LIN {X 0,Y 300.031,Z 474.405,A -85,B 0,C 180,E1 -16672.737,E2 -16672.737} C_VEL
LIN {X 0,Y 302.31,Z 463.313,A -85,B 0,C 180,E1 -16674.577,E2 -16674.577} C_VEL
LIN {X 0,Y 303.513,Z 452.468,A -85,B 0,C 180,E1 -16676.262,E2 -16676.262} C_VEL
LIN {X 0,Y 303.68,Z 440.033,A -85,B 0,C 180,E1 -16678.173,E2 -16678.173} C_VEL
LIN {X 0,Y 303.07,Z 428.896,A -85,B 0,C 180,E1 -16679.914,E2 -16679.914} C_VEL
LIN {X 0,Y 301.506,Z 416.977,A -85,B 0,C 180,E1 -16681.946,E2 -16681.946} C_VEL
LIN {X 0,Y 300.427,Z 410.712,A -85,B 0,C 180,E1 -16683.112,E2 -16683.112} C_VEL
LIN {X 0,Y 299.765,Z 406.041,A -85,B 0,C 180,E1 -16683.974,E2 -16683.974} C_VEL
LIN {X 0,Y 298.458,Z 400.385,A -85,B 0,C 180,E1 -16685.221,E2 -16685.221} C_VEL
LIN {X 0,Y 298.188,Z 398.22,A -85,B 0,C 180,E1 -16685.654,E2 -16685.654} C_VEL
LIN {X 0,Y 296.755,Z 392.365,A -85,B 0,C 180,E1 -16687.15,E2 -16687.15} C_VEL
LIN {X 0,Y 296.569,Z 389.678,A -85,B 0,C 180,E1 -16687.712,E2 -16687.712} C_VEL
LIN {X 0,Y 297.108,Z 387.807,A -85,B 0,C 180,E1 -16688.684,E2 -16688.684} C_VEL
LIN {X 0,Y 296.56,Z 383.262,A -85,B 0,C 180,E1 -16691.572,E2 -16691.572} C_VEL
LIN {X 0,Y 295.752,Z 379.256,A -85,B 0,C 180,E1 -16694.529,E2 -16694.529} C_VEL
LIN {X 0,Y 294.903,Z 375.161,A -85,B 0,C 180,E1 -16698.142,E2 -16698.142} C_VEL
LIN {X 0,Y 294.504,Z 373.34,A -85,B 0,C 180,E1 -16700.14,E2 -16700.14} C_VEL
LIN {X 0,Y 295.68,Z 374.442,A -85,B 0,C 180,E1 -16701.83,E2 -16701.83} C_VEL
LIN {X 0,Y 298.13,Z 375.151,A -85,B 0,C 180,E1 -16703.889,E2 -16703.889} C_VEL
LIN {X 0,Y 300.781,Z 377.325,A -85,B 0,C 180,E1 -16705.89,E2 -16705.89} C_VEL
LIN {X 0,Y 303.781,Z 380.298,A -85,B 0,C 180,E1 -16707.852,E2 -16707.852} C_VEL
LIN {X 0,Y 306.859,Z 384.143,A -85,B 0,C 180,E1 -16709.744,E2 -16709.744} C_VEL
LIN {X 0,Y 308.626,Z 387.569,A -85,B 0,C 180,E1 -16710.989,E2 -16710.989} C_VEL
LIN {X 0,Y 311.017,Z 394.757,A -85,B 0,C 180,E1 -16713.132,E2 -16713.132} C_VEL
LIN {X 0,Y 312.633,Z 402.039,A -85,B 0,C 180,E1 -16715.127,E2 -16715.127} C_VEL
LIN {X 0,Y 312.849,Z 403.656,A -85,B 0,C 180,E1 -16715.556,E2 -16715.556} C_VEL
LIN {X 0,Y 312.16,Z 406.591,A -85,B 0,C 180,E1 -16716.093,E2 -16716.093} C_VEL
LIN {X 0,Y 308.955,Z 416.302,A -85,B 0,C 180,E1 -16717.955,E2 -16717.955} C_VEL
LIN {X 0,Y 305.609,Z 425.337,A -85,B 0,C 180,E1 -16720.172,E2 -16720.172} C_VEL
LIN {X 0,Y 303.022,Z 431.501,A -85,B 0,C 180,E1 -16722.067,E2 -16722.067} C_VEL
LIN {X 0,Y 300.27,Z 437.333,A -85,B 0,C 180,E1 -16724.385,E2 -16724.385} C_VEL
LIN {X 0,Y 298.323,Z 441.092,A -85,B 0,C 180,E1 -16726.374,E2 -16726.374} C_VEL
LIN {X 0,Y 297.094,Z 443.088,A -85,B 0,C 180,E1 -16727.707,E2 -16727.707} C_VEL
LIN {X 0,Y 296.038,Z 444.641,A -85,B 0,C 180,E1 -16729.052,E2 -16729.052} C_VEL
LIN {X 0,Y 294.259,Z 446.525,A -85,B 0,C 180,E1 -16731.761,E2 -16731.761} C_VEL
LIN {X 0,Y 293.551,Z 446.906,A -85,B 0,C 180,E1 -16733.125,E2 -16733.125} C_VEL
LIN {X 0,Y 292.972,Z 446.863,A -85,B 0,C 180,E1 -16734.494,E2 -16734.494} C_VEL
LIN {X 0,Y 292.076,Z 445.605,A -85,B 0,C 180,E1 -16737.241,E2 -16737.241} C_VEL
LIN {X 0,Y 291.848,Z 444.386,A -85,B 0,C 180,E1 -16738.62,E2 -16738.62} C_VEL
LIN {X 0,Y 291.592,Z 441.785,A -85,B 0,C 180,E1 -16740.69,E2 -16740.69} C_VEL
LIN {X 0,Y 291.444,Z 438.224,A -85,B 0,C 180,E1 -16742.764,E2 -16742.764} C_VEL
LIN {X 0,Y 291.319,Z 435.273,A -85,B 0,C 180,E1 -16744.15,E2 -16744.15} C_VEL
LIN {X 0,Y 291.852,Z 429.89,A -85,B 0,C 180,E1 -16746.221,E2 -16746.221} C_VEL
LIN {X 0,Y 292.35,Z 422.074,A -85,B 0,C 180,E1 -16748.641,E2 -16748.641} C_VEL
LIN {X 0,Y 293.021,Z 413.88,A -85,B 0,C 180,E1 -16750.677,E2 -16750.677} C_VEL
LIN {X 0,Y 293.763,Z 403.548,A -85,B 0,C 180,E1 -16752.785,E2 -16752.785} C_VEL
LIN {X 0,Y 294.713,Z 393.16,A -85,B 0,C 180,E1 -16754.501,E2 -16754.501} C_VEL
LIN {X 0,Y 295.536,Z 381.754,A -85,B 0,C 180,E1 -16756.048,E2 -16756.048} C_VEL
LIN {X 0,Y 295.769,Z 377.353,A -85,B 0,C 180,E1 -16756.567,E2 -16756.567} C_VEL
LIN {X 0,Y 293.177,Z 366.301,A -85,B 0,C 180,E1 -16757.828,E2 -16757.828} C_VEL
LIN {X 0,Y 291.511,Z 359.165,A -85,B 0,C 180,E1 -16758.538,E2 -16758.538} C_VEL
LIN {X 0,Y 291.436,Z 359.181,A -85,B 0,C 180,E1 -16763.598,E2 -16763.598} C_VEL
LIN {X 0,Y 291.425,Z 359.184,A -85,B 0,C 180,E1 -16767.271,E2 -16767.271} C_VEL
LIN {X 0,Y 291.339,Z 359.193,A -85,B 0,C 180,E1 -16770.436,E2 -16770.436} C_VEL
LIN {X 0,Y 291.347,Z 359.19,A -85,B 0,C 180,E1 -16773.698,E2 -16773.698} C_VEL
LIN {X 0,Y 291.4,Z 359.186,A -85,B 0,C 180,E1 -16777.26,E2 -16777.26} C_VEL
LIN {X 0,Y 291.378,Z 359.19,A -85,B 0,C 180,E1 -16780.635,E2 -16780.635} C_VEL
LIN {X 0,Y 291.325,Z 359.195,A -85,B 0,C 180,E1 -16784.395,E2 -16784.395} C_VEL
LIN {X 0,Y 291.328,Z 359.196,A -85,B 0,C 180,E1 -16788.404,E2 -16788.404} C_VEL
LIN {X 0,Y 291.365,Z 359.189,A -85,B 0,C 180,E1 -16791.16,E2 -16791.16} C_VEL
LIN {X 0,Y 291.386,Z 359.191,A -85,B 0,C 180,E1 -16794.629,E2 -16794.629} C_VEL
LIN {X 0,Y 291.371,Z 359.189,A -85,B 0,C 180,E1 -16797.95,E2 -16797.95} C_VEL
LIN {X 0,Y 291.378,Z 359.187,A -85,B 0,C 180,E1 -16801.158,E2 -16801.158} C_VEL
LIN {X 0,Y 291.415,Z 359.186,A -85,B 0,C 180,E1 -16804.272,E2 -16804.272} C_VEL
LIN {X 0,Y 291.391,Z 359.185,A -85,B 0,C 180,E1 -16807.3,E2 -16807.3} C_VEL
LIN {X 0,Y 291.464,Z 359.18,A -85,B 0,C 180,E1 -16810.271,E2 -16810.271} C_VEL
LIN {X 0,Y 291.556,Z 359.167,A -85,B 0,C 180,E1 -16814.624,E2 -16814.624} C_VEL
LIN {X 0,Y 291.536,Z 359.167,A -85,B 0,C 180,E1 -16818.881,E2 -16818.881} C_VEL
LIN {X 0,Y 291.688,Z 359.15,A -85,B 0,C 180,E1 -16821.688,E2 -16821.688} C_VEL
LIN {X 0,Y 291.628,Z 359.157,A -85,B 0,C 180,E1 -16824.468,E2 -16824.468} C_VEL
LIN {X 0,Y 291.889,Z 359.124,A -85,B 0,C 180,E1 -16828.62,E2 -16828.62} C_VEL
LIN {X 0,Y 291.891,Z 359.124,A -85,B 0,C 180,E1 -16831.38,E2 -16831.38} C_VEL
LIN {X 0,Y 291.736,Z 359.142,A -85,B 0,C 180,E1 -16836.918,E2 -16836.918} C_VEL
LIN {X 0,Y 291.576,Z 359.166,A -85,B 0,C 180,E1 -16839.714,E2 -16839.714} C_VEL
LIN {X 0,Y 291.523,Z 359.172,A -85,B 0,C 180,E1 -16843.95,E2 -16843.95} C_VEL
LIN {X 0,Y 291.488,Z 359.173,A -85,B 0,C 180,E1 -16846.818,E2 -16846.818} C_VEL
LIN {X 0,Y 291.451,Z 359.18,A -85,B 0,C 180,E1 -16849.875,E2 -16849.875} C_VEL
LIN {X 0,Y 291.401,Z 359.185,A -85,B 0,C 180,E1 -16854.205,E2 -16854.205} C_VEL
LIN {X 0,Y 291.421,Z 359.184,A -85,B 0,C 180,E1 -16857.272,E2 -16857.272} C_VEL
LIN {X 0,Y 291.335,Z 359.191,A -85,B 0,C 180,E1 -16860.437,E2 -16860.437} C_VEL
LIN {X 0,Y 291.346,Z 359.194,A -85,B 0,C 180,E1 -16863.699,E2 -16863.699} C_VEL
LIN {X 0,Y 291.4,Z 359.188,A -85,B 0,C 180,E1 -16867.26,E2 -16867.26} C_VEL
LIN {X 0,Y 291.402,Z 359.184,A -85,B 0,C 180,E1 -16870.631,E2 -16870.631} C_VEL
LIN {X 0,Y 291.354,Z 359.19,A -85,B 0,C 180,E1 -16874.39,E2 -16874.39} C_VEL
LIN {X 0,Y 291.333,Z 359.192,A -85,B 0,C 180,E1 -16878.404,E2 -16878.404} C_VEL
LIN {X 0,Y 291.35,Z 359.196,A -85,B 0,C 180,E1 -16881.158,E2 -16881.158} C_VEL
LIN {X 0,Y 291.363,Z 359.19,A -85,B 0,C 180,E1 -16884.627,E2 -16884.627} C_VEL
LIN {X 0,Y 291.374,Z 359.187,A -85,B 0,C 180,E1 -16887.951,E2 -16887.951} C_VEL
LIN {X 0,Y 291.386,Z 359.189,A -85,B 0,C 180,E1 -16891.159,E2 -16891.159} C_VEL
LIN {X 0,Y 291.42,Z 359.181,A -85,B 0,C 180,E1 -16894.272,E2 -16894.272} C_VEL
LIN {X 0,Y 291.385,Z 359.188,A -85,B 0,C 180,E1 -16897.3,E2 -16897.3} C_VEL
LIN {X 0,Y 291.461,Z 359.177,A -85,B 0,C 180,E1 -16900.271,E2 -16900.271} C_VEL
LIN {X 0,Y 291.559,Z 359.168,A -85,B 0,C 180,E1 -16904.624,E2 -16904.624} C_VEL
LIN {X 0,Y 291.541,Z 359.17,A -85,B 0,C 180,E1 -16908.881,E2 -16908.881} C_VEL
LIN {X 0,Y 291.713,Z 359.144,A -85,B 0,C 180,E1 -16911.689,E2 -16911.689} C_VEL
LIN {X 0,Y 291.634,Z 359.159,A -85,B 0,C 180,E1 -16914.469,E2 -16914.469} C_VEL
LIN {X 0,Y 291.893,Z 359.126,A -85,B 0,C 180,E1 -16918.621,E2 -16918.621} C_VEL
LIN {X 0,Y 291.895,Z 359.122,A -85,B 0,C 180,E1 -16921.38,E2 -16921.38} C_VEL
LIN {X 0,Y 291.727,Z 359.144,A -85,B 0,C 180,E1 -16926.919,E2 -16926.919} C_VEL
LIN {X 0,Y 291.576,Z 359.162,A -85,B 0,C 180,E1 -16929.714,E2 -16929.714} C_VEL
LIN {X 0,Y 291.526,Z 359.168,A -85,B 0,C 180,E1 -16931.342,E2 -16931.342} C_VEL
LIN {X 0,Y 290.829,Z 359.259,A -85,B 0,C 180,E1 -16932.496,E2 -16932.496} C_VEL
LIN {X 0,Y 287.986,Z 359.613,A -85,B 0,C 180,E1 -16934.375,E2 -16934.375} C_VEL
LIN {X 0,Y 285.575,Z 359.913,A -85,B 0,C 180,E1 -16935.9,E2 -16935.9} C_VEL
LIN {X 0,Y 284.515,Z 360.041,A -85,B 0,C 180,E1 -16937.081,E2 -16937.081} C_VEL
LIN {X 0,Y 284.414,Z 360.052,A -85,B 0,C 180,E1 -16937.481,E2 -16937.481} C_VEL
LIN {X 0,Y 284.383,Z 360.063,A -85,B 0,C 180,E1 -16940.242,E2 -16940.242} C_VEL
LIN {X 0,Y 284.373,Z 360.062,A -85,B 0,C 180,E1 -16943.876,E2 -16943.876} C_VEL
LIN {X 0,Y 284.401,Z 360.055,A -85,B 0,C 180,E1 -16947.174,E2 -16947.174} C_VEL
LIN {X 0,Y 284.3,Z 360.069,A -85,B 0,C 180,E1 -16951.274,E2 -16951.274} C_VEL
LIN {X 0,Y 284.365,Z 360.061,A -85,B 0,C 180,E1 -16955.354,E2 -16955.354} C_VEL
LIN {X 0,Y 284.327,Z 360.068,A -85,B 0,C 180,E1 -16958.167,E2 -16958.167} C_VEL
LIN {X 0,Y 284.35,Z 360.119,A -85,B 0,C 180,E1 -16961.862,E2 -16961.862} C_VEL
LIN {X 0,Y 285.952,Z 368.508,A -85,B 0,C 180,E1 -16966.021,E2 -16966.021} C_VEL
LIN {X 0,Y 287.637,Z 376.818,A -85,B 0,C 180,E1 -16969.956,E2 -16969.956} C_VEL
LIN {X 0,Y 288.32,Z 381.031,A -85,B 0,C 180,E1 -16971.889,E2 -16971.889} C_VEL
LIN {X 0,Y 287.289,Z 387.971,A -85,B 0,C 180,E1 -16974.908,E2 -16974.908} C_VEL
LIN {X 0,Y 285.874,Z 397.284,A -85,B 0,C 180,E1 -16978.917,E2 -16978.917} C_VEL
LIN {X 0,Y 284.593,Z 408.243,A -85,B 0,C 180,E1 -16983.608,E2 -16983.608} C_VEL
LIN {X 0,Y 283.665,Z 419.379,A -85,B 0,C 180,E1 -16988.374,E2 -16988.374} C_VEL
LIN {X 0,Y 284.085,Z 432.923,A -85,B 0,C 180,E1 -16989.168,E2 -16989.168} C_VEL
LIN {X 0,Y 284.692,Z 446.489,A -85,B 0,C 180,E1 -16990.251,E2 -16990.251} C_VEL
LIN {X 0,Y 285.479,Z 460.384,A -85,B 0,C 180,E1 -16991.706,E2 -16991.706} C_VEL
LIN {X 0,Y 286.008,Z 471.143,A -85,B 0,C 180,E1 -16993.105,E2 -16993.105} C_VEL
LIN {X 0,Y 285.619,Z 477.09,A -85,B 0,C 180,E1 -16994.016,E2 -16994.016} C_VEL
LIN {X 0,Y 284.793,Z 486.616,A -85,B 0,C 180,E1 -16995.713,E2 -16995.713} C_VEL
LIN {X 0,Y 284.282,Z 494.949,A -85,B 0,C 180,E1 -16997.507,E2 -16997.507} C_VEL
LIN {X 0,Y 283.889,Z 503.067,A -85,B 0,C 180,E1 -16999.66,E2 -16999.66} C_VEL
LIN {X 0,Y 283.879,Z 510.11,A -85,B 0,C 180,E1 -17002.007,E2 -17002.007} C_VEL
LIN {X 0,Y 284.172,Z 515.473,A -85,B 0,C 180,E1 -17004.323,E2 -17004.323} C_VEL
LIN {X 0,Y 284.473,Z 519.112,A -85,B 0,C 180,E1 -17006.459,E2 -17006.459} C_VEL
LIN {X 0,Y 284.734,Z 521.591,A -85,B 0,C 180,E1 -17008.586,E2 -17008.586} C_VEL
LIN {X 0,Y 284.939,Z 522.63,A -85,B 0,C 180,E1 -17010,E2 -17010} C_VEL
LIN {X 0,Y 284.508,Z 523.101,A -85,B 0,C 180,E1 -17011.415,E2 -17011.415} C_VEL
LIN {X 0,Y 283.776,Z 522.795,A -85,B 0,C 180,E1 -17014.261,E2 -17014.261} C_VEL
LIN {X 0,Y 283.234,Z 520.886,A -85,B 0,C 180,E1 -17017.002,E2 -17017.002} C_VEL
LIN {X 0,Y 283.044,Z 518.199,A -85,B 0,C 180,E1 -17019.288,E2 -17019.288} C_VEL
LIN {X 0,Y 283.523,Z 513.371,A -85,B 0,C 180,E1 -17022.163,E2 -17022.163} C_VEL
LIN {X 0,Y 284.82,Z 506.896,A -85,B 0,C 180,E1 -17025.016,E2 -17025.016} C_VEL
LIN {X 0,Y 286.666,Z 499.719,A -85,B 0,C 180,E1 -17027.477,E2 -17027.477} C_VEL
LIN {X 0,Y 289.388,Z 491.01,A -85,B 0,C 180,E1 -17029.877,E2 -17029.877} C_VEL
LIN {X 0,Y 291.945,Z 482.139,A -85,B 0,C 180,E1 -17031.909,E2 -17031.909} C_VEL
LIN {X 0,Y 294.468,Z 471.795,A -85,B 0,C 180,E1 -17033.937,E2 -17033.937} C_VEL
LIN {X 0,Y 296.624,Z 461.632,A -85,B 0,C 180,E1 -17035.679,E2 -17035.679} C_VEL
LIN {X 0,Y 297.814,Z 450.071,A -85,B 0,C 180,E1 -17037.589,E2 -17037.589} C_VEL
LIN {X 0,Y 298.028,Z 437.389,A -85,B 0,C 180,E1 -17039.684,E2 -17039.684} C_VEL
LIN {X 0,Y 297.318,Z 425.925,A -85,B 0,C 180,E1 -17041.682,E2 -17041.682} C_VEL
LIN {X 0,Y 296.145,Z 415.72,A -85,B 0,C 180,E1 -17043.636,E2 -17043.636} C_VEL
LIN {X 0,Y 295.085,Z 408.633,A -85,B 0,C 180,E1 -17045.142,E2 -17045.142} C_VEL
LIN {X 0,Y 294.416,Z 403.054,A -85,B 0,C 180,E1 -17046.359,E2 -17046.359} C_VEL
LIN {X 0,Y 293.422,Z 397.739,A -85,B 0,C 180,E1 -17047.776,E2 -17047.776} C_VEL
LIN {X 0,Y 293.175,Z 394.527,A -85,B 0,C 180,E1 -17048.556,E2 -17048.556} C_VEL
LIN {X 0,Y 292.293,Z 391.653,A -85,B 0,C 180,E1 -17049.698,E2 -17049.698} C_VEL
LIN {X 0,Y 290.67,Z 386.21,A -85,B 0,C 180,E1 -17052.61,E2 -17052.61} C_VEL
LIN {X 0,Y 290.204,Z 383.651,A -85,B 0,C 180,E1 -17054.613,E2 -17054.613} C_VEL
LIN {X 0,Y 290.482,Z 381.502,A -85,B 0,C 180,E1 -17057.356,E2 -17057.356} C_VEL
LIN {X 0,Y 292.166,Z 380.152,A -85,B 0,C 180,E1 -17060.332,E2 -17060.332} C_VEL
LIN {X 0,Y 293.486,Z 381.114,A -85,B 0,C 180,E1 -17062.208,E2 -17062.208} C_VEL
LIN {X 0,Y 294.854,Z 381.369,A -85,B 0,C 180,E1 -17063.424,E2 -17063.424} C_VEL
LIN {X 0,Y 297.578,Z 383.63,A -85,B 0,C 180,E1 -17065.752,E2 -17065.752} C_VEL
LIN {X 0,Y 299.931,Z 386.143,A -85,B 0,C 180,E1 -17067.518,E2 -17067.518} C_VEL
LIN {X 0,Y 302.454,Z 389.396,A -85,B 0,C 180,E1 -17069.29,E2 -17069.29} C_VEL
LIN {X 0,Y 304.006,Z 392.328,A -85,B 0,C 180,E1 -17070.505,E2 -17070.505} C_VEL
LIN {X 0,Y 305.923,Z 399.005,A -85,B 0,C 180,E1 -17072.647,E2 -17072.647} C_VEL
LIN {X 0,Y 307.232,Z 406.151,A -85,B 0,C 180,E1 -17074.753,E2 -17074.753} C_VEL
LIN {X 0,Y 307.06,Z 408.046,A -85,B 0,C 180,E1 -17075.205,E2 -17075.205} C_VEL
LIN {X 0,Y 304.021,Z 416.608,A -85,B 0,C 180,E1 -17076.859,E2 -17076.859} C_VEL
LIN {X 0,Y 300.855,Z 424.65,A -85,B 0,C 180,E1 -17078.772,E2 -17078.772} C_VEL
LIN {X 0,Y 297.983,Z 431.197,A -85,B 0,C 180,E1 -17080.719,E2 -17080.719} C_VEL
LIN {X 0,Y 295.341,Z 436.536,A -85,B 0,C 180,E1 -17082.695,E2 -17082.695} C_VEL
LIN {X 0,Y 293.066,Z 440.748,A -85,B 0,C 180,E1 -17084.705,E2 -17084.705} C_VEL
LIN {X 0,Y 291.701,Z 443.029,A -85,B 0,C 180,E1 -17086.058,E2 -17086.058} C_VEL
LIN {X 0,Y 290.39,Z 444.878,A -85,B 0,C 180,E1 -17087.419,E2 -17087.419} C_VEL
LIN {X 0,Y 288.333,Z 447.305,A -85,B 0,C 180,E1 -17090.176,E2 -17090.176} C_VEL
LIN {X 0,Y 287.388,Z 447.971,A -85,B 0,C 180,E1 -17091.562,E2 -17091.562} C_VEL
LIN {X 0,Y 286.026,Z 448.048,A -85,B 0,C 180,E1 -17094.359,E2 -17094.359} C_VEL
LIN {X 0,Y 285.062,Z 446.608,A -85,B 0,C 180,E1 -17097.173,E2 -17097.173} C_VEL
LIN {X 0,Y 284.681,Z 443.497,A -85,B 0,C 180,E1 -17100,E2 -17100} C_VEL
LIN {X 0,Y 284.458,Z 440.106,A -85,B 0,C 180,E1 -17102.124,E2 -17102.124} C_VEL
LIN {X 0,Y 284.257,Z 435.712,A -85,B 0,C 180,E1 -17104.253,E2 -17104.253} C_VEL
LIN {X 0,Y 284.802,Z 430.166,A -85,B 0,C 180,E1 -17106.375,E2 -17106.375} C_VEL
LIN {X 0,Y 285.217,Z 423.367,A -85,B 0,C 180,E1 -17108.502,E2 -17108.502} C_VEL
LIN {X 0,Y 285.882,Z 415.183,A -85,B 0,C 180,E1 -17110.593,E2 -17110.593} C_VEL
LIN {X 0,Y 286.644,Z 404.889,A -85,B 0,C 180,E1 -17112.748,E2 -17112.748} C_VEL
LIN {X 0,Y 287.628,Z 394.593,A -85,B 0,C 180,E1 -17114.504,E2 -17114.504} C_VEL
LIN {X 0,Y 288.535,Z 381.958,A -85,B 0,C 180,E1 -17116.267,E2 -17116.267} C_VEL
LIN {X 0,Y 288.781,Z 379.024,A -85,B 0,C 180,E1 -17116.616,E2 -17116.616} C_VEL
LIN {X 0,Y 286.137,Z 367.424,A -85,B 0,C 180,E1 -17117.971,E2 -17117.971} C_VEL
LIN {X 0,Y 284.465,Z 360.045,A -85,B 0,C 180,E1 -17118.734,E2 -17118.734} C_VEL
LIN {X 0,Y 284.372,Z 360.059,A -85,B 0,C 180,E1 -17123.875,E2 -17123.875} C_VEL
LIN {X 0,Y 284.399,Z 360.06,A -85,B 0,C 180,E1 -17127.173,E2 -17127.173} C_VEL
LIN {X 0,Y 284.298,Z 360.071,A -85,B 0,C 180,E1 -17131.274,E2 -17131.274} C_VEL
LIN {X 0,Y 284.363,Z 360.062,A -85,B 0,C 180,E1 -17135.354,E2 -17135.354} C_VEL
LIN {X 0,Y 284.331,Z 360.065,A -85,B 0,C 180,E1 -17138.166,E2 -17138.166} C_VEL
LIN {X 0,Y 284.304,Z 360.067,A -85,B 0,C 180,E1 -17141.87,E2 -17141.87} C_VEL
LIN {X 0,Y 284.266,Z 360.073,A -85,B 0,C 180,E1 -17145.805,E2 -17145.805} C_VEL
LIN {X 0,Y 284.308,Z 360.068,A -85,B 0,C 180,E1 -17150.024,E2 -17150.024} C_VEL
LIN {X 0,Y 284.351,Z 360.062,A -85,B 0,C 180,E1 -17153.617,E2 -17153.617} C_VEL
LIN {X 0,Y 284.308,Z 360.068,A -85,B 0,C 180,E1 -17157.189,E2 -17157.189} C_VEL
LIN {X 0,Y 284.356,Z 360.065,A -85,B 0,C 180,E1 -17160.376,E2 -17160.376} C_VEL
LIN {X 0,Y 284.377,Z 360.059,A -85,B 0,C 180,E1 -17163.586,E2 -17163.586} C_VEL
LIN {X 0,Y 284.37,Z 360.062,A -85,B 0,C 180,E1 -17166.707,E2 -17166.707} C_VEL
LIN {X 0,Y 284.407,Z 360.055,A -85,B 0,C 180,E1 -17171.262,E2 -17171.262} C_VEL
LIN {X 0,Y 284.493,Z 360.048,A -85,B 0,C 180,E1 -17174.459,E2 -17174.459} C_VEL
LIN {X 0,Y 284.488,Z 360.047,A -85,B 0,C 180,E1 -17178.601,E2 -17178.601} C_VEL
LIN {X 0,Y 284.64,Z 360.027,A -85,B 0,C 180,E1 -17181.481,E2 -17181.481} C_VEL
LIN {X 0,Y 284.598,Z 360.034,A -85,B 0,C 180,E1 -17184.331,E2 -17184.331} C_VEL
LIN {X 0,Y 284.856,Z 360,A -85,B 0,C 180,E1 -17188.586,E2 -17188.586} C_VEL
LIN {X 0,Y 284.857,Z 360,A -85,B 0,C 180,E1 -17191.414,E2 -17191.414} C_VEL
LIN {X 0,Y 284.687,Z 360.02,A -85,B 0,C 180,E1 -17197.09,E2 -17197.09} C_VEL
LIN {X 0,Y 284.52,Z 360.045,A -85,B 0,C 180,E1 -17199.957,E2 -17199.957} C_VEL
LIN {X 0,Y 284.482,Z 360.047,A -85,B 0,C 180,E1 -17204.303,E2 -17204.303} C_VEL
LIN {X 0,Y 284.426,Z 360.054,A -85,B 0,C 180,E1 -17207.249,E2 -17207.249} C_VEL
LIN {X 0,Y 284.381,Z 360.059,A -85,B 0,C 180,E1 -17210.242,E2 -17210.242} C_VEL
LIN {X 0,Y 284.37,Z 360.063,A -85,B 0,C 180,E1 -17213.876,E2 -17213.876} C_VEL
LIN {X 0,Y 284.396,Z 360.059,A -85,B 0,C 180,E1 -17217.173,E2 -17217.173} C_VEL
LIN {X 0,Y 284.295,Z 360.072,A -85,B 0,C 180,E1 -17221.275,E2 -17221.275} C_VEL
LIN {X 0,Y 284.363,Z 360.066,A -85,B 0,C 180,E1 -17225.354,E2 -17225.354} C_VEL
LIN {X 0,Y 284.333,Z 360.064,A -85,B 0,C 180,E1 -17228.166,E2 -17228.166} C_VEL
LIN {X 0,Y 284.342,Z 360.064,A -85,B 0,C 180,E1 -17232.141,E2 -17232.141} C_VEL
LIN {X 0,Y 284.298,Z 360.068,A -85,B 0,C 180,E1 -17236.198,E2 -17236.198} C_VEL
LIN {X 0,Y 284.308,Z 360.068,A -85,B 0,C 180,E1 -17240.024,E2 -17240.024} C_VEL
LIN {X 0,Y 284.333,Z 360.065,A -85,B 0,C 180,E1 -17243.614,E2 -17243.614} C_VEL
LIN {X 0,Y 284.31,Z 360.071,A -85,B 0,C 180,E1 -17247.19,E2 -17247.19} C_VEL
LIN {X 0,Y 284.362,Z 360.062,A -85,B 0,C 180,E1 -17250.377,E2 -17250.377} C_VEL
LIN {X 0,Y 284.381,Z 360.058,A -85,B 0,C 180,E1 -17253.587,E2 -17253.587} C_VEL
LIN {X 0,Y 284.37,Z 360.063,A -85,B 0,C 180,E1 -17256.707,E2 -17256.707} C_VEL
LIN {X 0,Y 284.407,Z 360.056,A -85,B 0,C 180,E1 -17261.262,E2 -17261.262} C_VEL
LIN {X 0,Y 284.496,Z 360.046,A -85,B 0,C 180,E1 -17264.459,E2 -17264.459} C_VEL
LIN {X 0,Y 284.493,Z 360.049,A -85,B 0,C 180,E1 -17268.602,E2 -17268.602} C_VEL
LIN {X 0,Y 284.663,Z 360.022,A -85,B 0,C 180,E1 -17271.481,E2 -17271.481} C_VEL
LIN {X 0,Y 284.605,Z 360.033,A -85,B 0,C 180,E1 -17274.332,E2 -17274.332} C_VEL
LIN {X 0,Y 284.859,Z 360.003,A -85,B 0,C 180,E1 -17278.586,E2 -17278.586} C_VEL
LIN {X 0,Y 284.861,Z 359.998,A -85,B 0,C 180,E1 -17281.414,E2 -17281.414} C_VEL
LIN {X 0,Y 284.678,Z 360.021,A -85,B 0,C 180,E1 -17287.091,E2 -17287.091} C_VEL
LIN {X 0,Y 284.521,Z 360.042,A -85,B 0,C 180,E1 -17289.957,E2 -17289.957} C_VEL
LIN {X 0,Y 284.486,Z 360.05,A -85,B 0,C 180,E1 -17294.303,E2 -17294.303} C_VEL
LIN {X 0,Y 284.414,Z 360.052,A -85,B 0,C 180,E1 -17297.481,E2 -17297.481} C_VEL
LIN {X 0,Y 283.687,Z 360.147,A -85,B 0,C 180,E1 -17298.662,E2 -17298.662} C_VEL
LIN {X 0,Y 280.765,Z 360.511,A -85,B 0,C 180,E1 -17300.583,E2 -17300.583} C_VEL
LIN {X 0,Y 278.351,Z 360.815,A -85,B 0,C 180,E1 -17302.145,E2 -17302.145} C_VEL
LIN {X 0,Y 277.371,Z 360.933,A -85,B 0,C 180,E1 -17303.356,E2 -17303.356} C_VEL
LIN {X 0,Y 277.319,Z 360.94,A -85,B 0,C 180,E1 -17303.765,E2 -17303.765} C_VEL
LIN {X 0,Y 277.33,Z 360.937,A -85,B 0,C 180,E1 -17307.505,E2 -17307.505} C_VEL
LIN {X 0,Y 277.275,Z 360.945,A -85,B 0,C 180,E1 -17310.481,E2 -17310.481} C_VEL
LIN {X 0,Y 277.258,Z 360.949,A -85,B 0,C 180,E1 -17313.895,E2 -17313.895} C_VEL
LIN {X 0,Y 277.284,Z 360.944,A -85,B 0,C 180,E1 -17317.467,E2 -17317.467} C_VEL
LIN {X 0,Y 277.314,Z 361.062,A -85,B 0,C 180,E1 -17321.702,E2 -17321.702} C_VEL
LIN {X 0,Y 278.879,Z 369.353,A -85,B 0,C 180,E1 -17325.907,E2 -17325.907} C_VEL
LIN {X 0,Y 280.674,Z 378.095,A -85,B 0,C 180,E1 -17330.149,E2 -17330.149} C_VEL
LIN {X 0,Y 281.253,Z 381.599,A -85,B 0,C 180,E1 -17331.796,E2 -17331.796} C_VEL
LIN {X 0,Y 280.228,Z 388.25,A -85,B 0,C 180,E1 -17334.772,E2 -17334.772} C_VEL
LIN {X 0,Y 278.742,Z 397.811,A -85,B 0,C 180,E1 -17339.01,E2 -17339.01} C_VEL
LIN {X 0,Y 277.467,Z 408.383,A -85,B 0,C 180,E1 -17343.688,E2 -17343.688} C_VEL
LIN {X 0,Y 276.606,Z 418.489,A -85,B 0,C 180,E1 -17348.137,E2 -17348.137} C_VEL
LIN {X 0,Y 276.996,Z 432.602,A -85,B 0,C 180,E1 -17348.999,E2 -17348.999} C_VEL
LIN {X 0,Y 277.619,Z 446.296,A -85,B 0,C 180,E1 -17350.146,E2 -17350.146} C_VEL
LIN {X 0,Y 278.348,Z 459.692,A -85,B 0,C 180,E1 -17351.602,E2 -17351.602} C_VEL
LIN {X 0,Y 278.929,Z 471.618,A -85,B 0,C 180,E1 -17353.23,E2 -17353.23} C_VEL
LIN {X 0,Y 278.293,Z 480.051,A -85,B 0,C 180,E1 -17354.623,E2 -17354.623} C_VEL
LIN {X 0,Y 277.499,Z 489.237,A -85,B 0,C 180,E1 -17356.451,E2 -17356.451} C_VEL
LIN {X 0,Y 277.067,Z 496.903,A -85,B 0,C 180,E1 -17358.292,E2 -17358.292} C_VEL
LIN {X 0,Y 276.839,Z 504.435,A -85,B 0,C 180,E1 -17360.502,E2 -17360.502} C_VEL
LIN {X 0,Y 276.984,Z 510.428,A -85,B 0,C 180,E1 -17362.711,E2 -17362.711} C_VEL
LIN {X 0,Y 277.325,Z 515.088,A -85,B 0,C 180,E1 -17364.911,E2 -17364.911} C_VEL
LIN {X 0,Y 277.602,Z 518.473,A -85,B 0,C 180,E1 -17367.098,E2 -17367.098} C_VEL
LIN {X 0,Y 277.765,Z 520.094,A -85,B 0,C 180,E1 -17368.55,E2 -17368.55} C_VEL
LIN {X 0,Y 277.979,Z 521.259,A -85,B 0,C 180,E1 -17370,E2 -17370} C_VEL
LIN {X 0,Y 277.513,Z 521.797,A -85,B 0,C 180,E1 -17371.451,E2 -17371.451} C_VEL
LIN {X 0,Y 276.72,Z 521.616,A -85,B 0,C 180,E1 -17374.37,E2 -17374.37} C_VEL
LIN {X 0,Y 276.185,Z 520.013,A -85,B 0,C 180,E1 -17377.056,E2 -17377.056} C_VEL
LIN {X 0,Y 275.99,Z 518.267,A -85,B 0,C 180,E1 -17378.788,E2 -17378.788} C_VEL
LIN {X 0,Y 276.272,Z 514.056,A -85,B 0,C 180,E1 -17381.742,E2 -17381.742} C_VEL
LIN {X 0,Y 277.461,Z 508.279,A -85,B 0,C 180,E1 -17384.673,E2 -17384.673} C_VEL
LIN {X 0,Y 278.915,Z 502.744,A -85,B 0,C 180,E1 -17386.87,E2 -17386.87} C_VEL
LIN {X 0,Y 281.405,Z 495.092,A -85,B 0,C 180,E1 -17389.324,E2 -17389.324} C_VEL
LIN {X 0,Y 284.613,Z 485.785,A -85,B 0,C 180,E1 -17391.74,E2 -17391.74} C_VEL
LIN {X 0,Y 287.136,Z 476.452,A -85,B 0,C 180,E1 -17393.82,E2 -17393.82} C_VEL
LIN {X 0,Y 289.943,Z 465.625,A -85,B 0,C 180,E1 -17395.869,E2 -17395.869} C_VEL
LIN {X 0,Y 291.624,Z 455.632,A -85,B 0,C 180,E1 -17397.64,E2 -17397.64} C_VEL
LIN {X 0,Y 292.514,Z 442.946,A -85,B 0,C 180,E1 -17399.874,E2 -17399.874} C_VEL
LIN {X 0,Y 292.417,Z 431.803,A -85,B 0,C 180,E1 -17401.921,E2 -17401.921} C_VEL
LIN {X 0,Y 291.662,Z 420.26,A -85,B 0,C 180,E1 -17404.244,E2 -17404.244} C_VEL
LIN {X 0,Y 291.026,Z 413.693,A -85,B 0,C 180,E1 -17405.706,E2 -17405.706} C_VEL
LIN {X 0,Y 290.426,Z 407.325,A -85,B 0,C 180,E1 -17407.227,E2 -17407.227} C_VEL
LIN {X 0,Y 289.842,Z 400.226,A -85,B 0,C 180,E1 -17409.111,E2 -17409.111} C_VEL
LIN {X 0,Y 289.088,Z 397.065,A -85,B 0,C 180,E1 -17410.429,E2 -17410.429} C_VEL
LIN {X 0,Y 287.944,Z 392.313,A -85,B 0,C 180,E1 -17413.111,E2 -17413.111} C_VEL
LIN {X 0,Y 287.634,Z 389.914,A -85,B 0,C 180,E1 -17415.12,E2 -17415.12} C_VEL
LIN {X 0,Y 287.826,Z 388.324,A -85,B 0,C 180,E1 -17417.099,E2 -17417.099} C_VEL
LIN {X 0,Y 288.593,Z 387.235,A -85,B 0,C 180,E1 -17419.02,E2 -17419.02} C_VEL
LIN {X 0,Y 289.737,Z 387.07,A -85,B 0,C 180,E1 -17420.915,E2 -17420.915} C_VEL
LIN {X 0,Y 291.316,Z 387.719,A -85,B 0,C 180,E1 -17422.906,E2 -17422.906} C_VEL
LIN {X 0,Y 293.314,Z 389.164,A -85,B 0,C 180,E1 -17424.896,E2 -17424.896} C_VEL
LIN {X 0,Y 296.118,Z 392.043,A -85,B 0,C 180,E1 -17427.29,E2 -17427.29} C_VEL
LIN {X 0,Y 298.876,Z 396.108,A -85,B 0,C 180,E1 -17429.567,E2 -17429.567} C_VEL
LIN {X 0,Y 300.093,Z 399.729,A -85,B 0,C 180,E1 -17430.964,E2 -17430.964} C_VEL
LIN {X 0,Y 301.268,Z 405.671,A -85,B 0,C 180,E1 -17432.928,E2 -17432.928} C_VEL
LIN {X 0,Y 301.733,Z 409.541,A -85,B 0,C 180,E1 -17434.149,E2 -17434.149} C_VEL
LIN {X 0,Y 301.576,Z 411.082,A -85,B 0,C 180,E1 -17434.549,E2 -17434.549} C_VEL
LIN {X 0,Y 298.061,Z 419.981,A -85,B 0,C 180,E1 -17436.369,E2 -17436.369} C_VEL
LIN {X 0,Y 294.649,Z 427.79,A -85,B 0,C 180,E1 -17438.376,E2 -17438.376} C_VEL
LIN {X 0,Y 291.712,Z 433.808,A -85,B 0,C 180,E1 -17440.288,E2 -17440.288} C_VEL
LIN {X 0,Y 288.928,Z 438.878,A -85,B 0,C 180,E1 -17442.298,E2 -17442.298} C_VEL
LIN {X 0,Y 286.541,Z 442.844,A -85,B 0,C 180,E1 -17444.348,E2 -17444.348} C_VEL
LIN {X 0,Y 285.087,Z 444.954,A -85,B 0,C 180,E1 -17445.728,E2 -17445.728} C_VEL
LIN {X 0,Y 282.523,Z 447.955,A -85,B 0,C 180,E1 -17448.521,E2 -17448.521} C_VEL
LIN {X 0,Y 281.523,Z 448.856,A -85,B 0,C 180,E1 -17449.936,E2 -17449.936} C_VEL
LIN {X 0,Y 279.722,Z 449.494,A -85,B 0,C 180,E1 -17452.783,E2 -17452.783} C_VEL
LIN {X 0,Y 278.451,Z 448.614,A -85,B 0,C 180,E1 -17455.657,E2 -17455.657} C_VEL
LIN {X 0,Y 277.804,Z 446.087,A -85,B 0,C 180,E1 -17458.55,E2 -17458.55} C_VEL
LIN {X 0,Y 277.463,Z 443.158,A -85,B 0,C 180,E1 -17460.725,E2 -17460.725} C_VEL
LIN {X 0,Y 277.292,Z 439.259,A -85,B 0,C 180,E1 -17462.905,E2 -17462.905} C_VEL
LIN {X 0,Y 277.2,Z 436.096,A -85,B 0,C 180,E1 -17464.362,E2 -17464.362} C_VEL
LIN {X 0,Y 277.814,Z 429.269,A -85,B 0,C 180,E1 -17466.901,E2 -17466.901} C_VEL
LIN {X 0,Y 278.426,Z 420.714,A -85,B 0,C 180,E1 -17469.443,E2 -17469.443} C_VEL
LIN {X 0,Y 279.156,Z 411.548,A -85,B 0,C 180,E1 -17471.619,E2 -17471.619} C_VEL
LIN {X 0,Y 279.979,Z 401.362,A -85,B 0,C 180,E1 -17473.611,E2 -17473.611} C_VEL
LIN {X 0,Y 281.003,Z 390.037,A -85,B 0,C 180,E1 -17475.41,E2 -17475.41} C_VEL
LIN {X 0,Y 281.609,Z 378.995,A -85,B 0,C 180,E1 -17476.865,E2 -17476.865} C_VEL
LIN {X 0,Y 278.782,Z 367.124,A -85,B 0,C 180,E1 -17478.263,E2 -17478.263} C_VEL
LIN {X 0,Y 277.423,Z 360.925,A -85,B 0,C 180,E1 -17478.892,E2 -17478.892} C_VEL
LIN {X 0,Y 277.322,Z 360.937,A -85,B 0,C 180,E1 -17484.17,E2 -17484.17} C_VEL
LIN {X 0,Y 277.328,Z 360.938,A -85,B 0,C 180,E1 -17487.505,E2 -17487.505} C_VEL
LIN {X 0,Y 277.273,Z 360.945,A -85,B 0,C 180,E1 -17490.481,E2 -17490.481} C_VEL
LIN {X 0,Y 277.256,Z 360.945,A -85,B 0,C 180,E1 -17493.894,E2 -17493.894} C_VEL
LIN {X 0,Y 277.287,Z 360.943,A -85,B 0,C 180,E1 -17497.466,E2 -17497.466} C_VEL
LIN {X 0,Y 277.242,Z 360.949,A -85,B 0,C 180,E1 -17501.23,E2 -17501.23} C_VEL
LIN {X 0,Y 277.221,Z 360.952,A -85,B 0,C 180,E1 -17505.222,E2 -17505.222} C_VEL
LIN {X 0,Y 277.224,Z 360.95,A -85,B 0,C 180,E1 -17509.512,E2 -17509.512} C_VEL
LIN {X 0,Y 277.283,Z 360.946,A -85,B 0,C 180,E1 -17512.533,E2 -17512.533} C_VEL
LIN {X 0,Y 277.255,Z 360.948,A -85,B 0,C 180,E1 -17516.105,E2 -17516.105} C_VEL
LIN {X 0,Y 277.262,Z 360.944,A -85,B 0,C 180,E1 -17519.538,E2 -17519.538} C_VEL
LIN {X 0,Y 277.357,Z 360.935,A -85,B 0,C 180,E1 -17522.864,E2 -17522.864} C_VEL
LIN {X 0,Y 277.33,Z 360.939,A -85,B 0,C 180,E1 -17526.08,E2 -17526.08} C_VEL
LIN {X 0,Y 277.347,Z 360.936,A -85,B 0,C 180,E1 -17530.766,E2 -17530.766} C_VEL
LIN {X 0,Y 277.435,Z 360.923,A -85,B 0,C 180,E1 -17535.326,E2 -17535.326} C_VEL
LIN {X 0,Y 277.462,Z 360.922,A -85,B 0,C 180,E1 -17539.787,E2 -17539.787} C_VEL
LIN {X 0,Y 277.642,Z 360.899,A -85,B 0,C 180,E1 -17542.729,E2 -17542.729} C_VEL
LIN {X 0,Y 277.822,Z 360.877,A -85,B 0,C 180,E1 -17548.551,E2 -17548.551} C_VEL
LIN {X 0,Y 277.823,Z 360.877,A -85,B 0,C 180,E1 -17551.45,E2 -17551.45} C_VEL
LIN {X 0,Y 277.642,Z 360.899,A -85,B 0,C 180,E1 -17557.271,E2 -17557.271} C_VEL
LIN {X 0,Y 277.462,Z 360.922,A -85,B 0,C 180,E1 -17560.213,E2 -17560.213} C_VEL
LIN {X 0,Y 277.435,Z 360.923,A -85,B 0,C 180,E1 -17564.674,E2 -17564.674} C_VEL
LIN {X 0,Y 277.346,Z 360.936,A -85,B 0,C 180,E1 -17569.234,E2 -17569.234} C_VEL
LIN {X 0,Y 277.33,Z 360.939,A -85,B 0,C 180,E1 -17573.921,E2 -17573.921} C_VEL
LIN {X 0,Y 277.324,Z 360.942,A -85,B 0,C 180,E1 -17577.505,E2 -17577.505} C_VEL
LIN {X 0,Y 277.273,Z 360.943,A -85,B 0,C 180,E1 -17580.482,E2 -17580.482} C_VEL
LIN {X 0,Y 277.255,Z 360.948,A -85,B 0,C 180,E1 -17583.895,E2 -17583.895} C_VEL
LIN {X 0,Y 277.288,Z 360.945,A -85,B 0,C 180,E1 -17587.467,E2 -17587.467} C_VEL
LIN {X 0,Y 277.294,Z 360.945,A -85,B 0,C 180,E1 -17591.222,E2 -17591.222} C_VEL
LIN {X 0,Y 277.244,Z 360.952,A -85,B 0,C 180,E1 -17595.218,E2 -17595.218} C_VEL
LIN {X 0,Y 277.227,Z 360.952,A -85,B 0,C 180,E1 -17599.512,E2 -17599.512} C_VEL
LIN {X 0,Y 277.267,Z 360.946,A -85,B 0,C 180,E1 -17602.531,E2 -17602.531} C_VEL
LIN {X 0,Y 277.249,Z 360.946,A -85,B 0,C 180,E1 -17606.105,E2 -17606.105} C_VEL
LIN {X 0,Y 277.264,Z 360.946,A -85,B 0,C 180,E1 -17609.539,E2 -17609.539} C_VEL
LIN {X 0,Y 277.362,Z 360.937,A -85,B 0,C 180,E1 -17612.865,E2 -17612.865} C_VEL
LIN {X 0,Y 277.332,Z 360.936,A -85,B 0,C 180,E1 -17616.08,E2 -17616.08} C_VEL
LIN {X 0,Y 277.349,Z 360.939,A -85,B 0,C 180,E1 -17620.767,E2 -17620.767} C_VEL
LIN {X 0,Y 277.438,Z 360.924,A -85,B 0,C 180,E1 -17625.326,E2 -17625.326} C_VEL
LIN {X 0,Y 277.511,Z 360.914,A -85,B 0,C 180,E1 -17629.789,E2 -17629.789} C_VEL
LIN {X 0,Y 277.658,Z 360.9,A -85,B 0,C 180,E1 -17632.729,E2 -17632.729} C_VEL
LIN {X 0,Y 277.825,Z 360.879,A -85,B 0,C 180,E1 -17638.551,E2 -17638.551} C_VEL
LIN {X 0,Y 277.826,Z 360.874,A -85,B 0,C 180,E1 -17641.45,E2 -17641.45} C_VEL
LIN {X 0,Y 277.632,Z 360.898,A -85,B 0,C 180,E1 -17647.272,E2 -17647.272} C_VEL
LIN {X 0,Y 277.464,Z 360.923,A -85,B 0,C 180,E1 -17650.213,E2 -17650.213} C_VEL
LIN {X 0,Y 277.439,Z 360.925,A -85,B 0,C 180,E1 -17654.674,E2 -17654.674} C_VEL
LIN {X 0,Y 277.349,Z 360.934,A -85,B 0,C 180,E1 -17659.234,E2 -17659.234} C_VEL
LIN {X 0,Y 277.319,Z 360.94,A -85,B 0,C 180,E1 -17663.765,E2 -17663.765} C_VEL
LIN {X 0,Y 276.713,Z 361.022,A -85,B 0,C 180,E1 -17664.979,E2 -17664.979} C_VEL
LIN {X 0,Y 273.829,Z 361.382,A -85,B 0,C 180,E1 -17666.953,E2 -17666.953} C_VEL
LIN {X 0,Y 271.339,Z 361.687,A -85,B 0,C 180,E1 -17668.558,E2 -17668.558} C_VEL
LIN {X 0,Y 270.27,Z 361.82,A -85,B 0,C 180,E1 -17669.804,E2 -17669.804} C_VEL
LIN {X 0,Y 270.186,Z 361.826,A -85,B 0,C 180,E1 -17670.226,E2 -17670.226} C_VEL
LIN {X 0,Y 270.224,Z 361.824,A -85,B 0,C 180,E1 -17673.668,E2 -17673.668} C_VEL
LIN {X 0,Y 270.241,Z 361.82,A -85,B 0,C 180,E1 -17676.738,E2 -17676.738} C_VEL
LIN {X 0,Y 270.258,Z 361.82,A -85,B 0,C 180,E1 -17681.426,E2 -17681.426} C_VEL
LIN {X 0,Y 271.794,Z 370.016,A -85,B 0,C 180,E1 -17685.72,E2 -17685.72} C_VEL
LIN {X 0,Y 273.722,Z 379.355,A -85,B 0,C 180,E1 -17690.379,E2 -17690.379} C_VEL
LIN {X 0,Y 274.137,Z 382.819,A -85,B 0,C 180,E1 -17692.027,E2 -17692.027} C_VEL
LIN {X 0,Y 272.559,Z 392.237,A -85,B 0,C 180,E1 -17696.351,E2 -17696.351} C_VEL
LIN {X 0,Y 270.955,Z 403.036,A -85,B 0,C 180,E1 -17701.285,E2 -17701.285} C_VEL
LIN {X 0,Y 269.936,Z 412.681,A -85,B 0,C 180,E1 -17705.68,E2 -17705.68} C_VEL
LIN {X 0,Y 269.554,Z 417.512,A -85,B 0,C 180,E1 -17707.887,E2 -17707.887} C_VEL
LIN {X 0,Y 269.925,Z 432.884,A -85,B 0,C 180,E1 -17708.888,E2 -17708.888} C_VEL
LIN {X 0,Y 270.501,Z 445.685,A -85,B 0,C 180,E1 -17710.016,E2 -17710.016} C_VEL
LIN {X 0,Y 271.214,Z 458.82,A -85,B 0,C 180,E1 -17711.492,E2 -17711.492} C_VEL
LIN {X 0,Y 271.789,Z 470.23,A -85,B 0,C 180,E1 -17713.09,E2 -17713.09} C_VEL
LIN {X 0,Y 271.633,Z 474.917,A -85,B 0,C 180,E1 -17713.851,E2 -17713.851} C_VEL
LIN {X 0,Y 270.751,Z 484.831,A -85,B 0,C 180,E1 -17715.724,E2 -17715.724} C_VEL
LIN {X 0,Y 270.225,Z 493.062,A -85,B 0,C 180,E1 -17717.61,E2 -17717.61} C_VEL
LIN {X 0,Y 269.904,Z 501.076,A -85,B 0,C 180,E1 -17719.877,E2 -17719.877} C_VEL
LIN {X 0,Y 269.975,Z 508.473,A -85,B 0,C 180,E1 -17722.521,E2 -17722.521} C_VEL
LIN {X 0,Y 270.317,Z 513.313,A -85,B 0,C 180,E1 -17724.779,E2 -17724.779} C_VEL
LIN {X 0,Y 270.64,Z 516.877,A -85,B 0,C 180,E1 -17727.023,E2 -17727.023} C_VEL
LIN {X 0,Y 270.815,Z 518.569,A -85,B 0,C 180,E1 -17728.513,E2 -17728.513} C_VEL
LIN {X 0,Y 271.01,Z 519.804,A -85,B 0,C 180,E1 -17730,E2 -17730} C_VEL
LIN {X 0,Y 270.515,Z 520.453,A -85,B 0,C 180,E1 -17731.489,E2 -17731.489} C_VEL
LIN {X 0,Y 270.045,Z 520.656,A -85,B 0,C 180,E1 -17732.984,E2 -17732.984} C_VEL
LIN {X 0,Y 269.663,Z 520.433,A -85,B 0,C 180,E1 -17734.484,E2 -17734.484} C_VEL
LIN {X 0,Y 269.131,Z 519.09,A -85,B 0,C 180,E1 -17737.102,E2 -17737.102} C_VEL
LIN {X 0,Y 268.922,Z 517.368,A -85,B 0,C 180,E1 -17739.021,E2 -17739.021} C_VEL
LIN {X 0,Y 269.261,Z 513.389,A -85,B 0,C 180,E1 -17742.053,E2 -17742.053} C_VEL
LIN {X 0,Y 270.549,Z 507.852,A -85,B 0,C 180,E1 -17745.056,E2 -17745.056} C_VEL
LIN {X 0,Y 272.381,Z 501.764,A -85,B 0,C 180,E1 -17747.61,E2 -17747.61} C_VEL
LIN {X 0,Y 275.145,Z 494.103,A -85,B 0,C 180,E1 -17750.171,E2 -17750.171} C_VEL
LIN {X 0,Y 278.48,Z 484.964,A -85,B 0,C 180,E1 -17752.635,E2 -17752.635} C_VEL
LIN {X 0,Y 281.294,Z 475.836,A -85,B 0,C 180,E1 -17754.739,E2 -17754.739} C_VEL
LIN {X 0,Y 284.145,Z 465.59,A -85,B 0,C 180,E1 -17756.79,E2 -17756.79} C_VEL
LIN {X 0,Y 285.919,Z 455.825,A -85,B 0,C 180,E1 -17758.641,E2 -17758.641} C_VEL
LIN {X 0,Y 287.107,Z 443.156,A -85,B 0,C 180,E1 -17761.045,E2 -17761.045} C_VEL
LIN {X 0,Y 287.278,Z 431.27,A -85,B 0,C 180,E1 -17763.429,E2 -17763.429} C_VEL
LIN {X 0,Y 286.89,Z 419.434,A -85,B 0,C 180,E1 -17766.059,E2 -17766.059} C_VEL
LIN {X 0,Y 286.549,Z 412.442,A -85,B 0,C 180,E1 -17767.819,E2 -17767.819} C_VEL
LIN {X 0,Y 286.32,Z 405.9,A -85,B 0,C 180,E1 -17769.658,E2 -17769.658} C_VEL
LIN {X 0,Y 285.76,Z 402.674,A -85,B 0,C 180,E1 -17771.024,E2 -17771.024} C_VEL
LIN {X 0,Y 284.959,Z 398.234,A -85,B 0,C 180,E1 -17773.676,E2 -17773.676} C_VEL
LIN {X 0,Y 284.829,Z 395.501,A -85,B 0,C 180,E1 -17776.299,E2 -17776.299} C_VEL
LIN {X 0,Y 285.337,Z 394.168,A -85,B 0,C 180,E1 -17778.315,E2 -17778.315} C_VEL
LIN {X 0,Y 286.359,Z 393.567,A -85,B 0,C 180,E1 -17780.349,E2 -17780.349} C_VEL
LIN {X 0,Y 287.681,Z 393.905,A -85,B 0,C 180,E1 -17782.356,E2 -17782.356} C_VEL
LIN {X 0,Y 289.419,Z 394.957,A -85,B 0,C 180,E1 -17784.352,E2 -17784.352} C_VEL
LIN {X 0,Y 292.369,Z 398.157,A -85,B 0,C 180,E1 -17787.282,E2 -17787.282} C_VEL
LIN {X 0,Y 294.407,Z 401.402,A -85,B 0,C 180,E1 -17789.248,E2 -17789.248} C_VEL
LIN {X 0,Y 295.248,Z 404.232,A -85,B 0,C 180,E1 -17790.441,E2 -17790.441} C_VEL
LIN {X 0,Y 296.175,Z 410.878,A -85,B 0,C 180,E1 -17792.813,E2 -17792.813} C_VEL
LIN {X 0,Y 296.316,Z 413.195,A -85,B 0,C 180,E1 -17793.595,E2 -17793.595} C_VEL
LIN {X 0,Y 296.004,Z 414.567,A -85,B 0,C 180,E1 -17793.944,E2 -17793.944} C_VEL
LIN {X 0,Y 292.164,Z 423.328,A -85,B 0,C 180,E1 -17795.862,E2 -17795.862} C_VEL
LIN {X 0,Y 288.692,Z 430.532,A -85,B 0,C 180,E1 -17797.831,E2 -17797.831} C_VEL
LIN {X 0,Y 285.467,Z 436.431,A -85,B 0,C 180,E1 -17799.838,E2 -17799.838} C_VEL
LIN {X 0,Y 282.551,Z 441.197,A -85,B 0,C 180,E1 -17801.885,E2 -17801.885} C_VEL
LIN {X 0,Y 280.021,Z 444.917,A -85,B 0,C 180,E1 -17803.973,E2 -17803.973} C_VEL
LIN {X 0,Y 277.012,Z 448.458,A -85,B 0,C 180,E1 -17806.801,E2 -17806.801} C_VEL
LIN {X 0,Y 275.771,Z 449.619,A -85,B 0,C 180,E1 -17808.236,E2 -17808.236} C_VEL
LIN {X 0,Y 273.638,Z 450.767,A -85,B 0,C 180,E1 -17811.135,E2 -17811.135} C_VEL
LIN {X 0,Y 272.126,Z 450.403,A -85,B 0,C 180,E1 -17814.07,E2 -17814.07} C_VEL
LIN {X 0,Y 271.452,Z 449.63,A -85,B 0,C 180,E1 -17815.545,E2 -17815.545} C_VEL
LIN {X 0,Y 270.758,Z 446.91,A -85,B 0,C 180,E1 -17818.512,E2 -17818.512} C_VEL
LIN {X 0,Y 270.401,Z 443.804,A -85,B 0,C 180,E1 -17820.744,E2 -17820.744} C_VEL
LIN {X 0,Y 270.213,Z 439.732,A -85,B 0,C 180,E1 -17822.982,E2 -17822.982} C_VEL
LIN {X 0,Y 270.387,Z 434.57,A -85,B 0,C 180,E1 -17825.219,E2 -17825.219} C_VEL
LIN {X 0,Y 270.799,Z 428.215,A -85,B 0,C 180,E1 -17827.456,E2 -17827.456} C_VEL
LIN {X 0,Y 271.375,Z 420.696,A -85,B 0,C 180,E1 -17829.629,E2 -17829.629} C_VEL
LIN {X 0,Y 272.164,Z 411.07,A -85,B 0,C 180,E1 -17831.922,E2 -17831.922} C_VEL
LIN {X 0,Y 273.082,Z 400.571,A -85,B 0,C 180,E1 -17833.962,E2 -17833.962} C_VEL
LIN {X 0,Y 274.055,Z 388.94,A -85,B 0,C 180,E1 -17835.811,E2 -17835.811} C_VEL
LIN {X 0,Y 274.589,Z 380.122,A -85,B 0,C 180,E1 -17836.975,E2 -17836.975} C_VEL
LIN {X 0,Y 271.651,Z 367.664,A -85,B 0,C 180,E1 -17838.477,E2 -17838.477} C_VEL
LIN {X 0,Y 270.369,Z 361.806,A -85,B 0,C 180,E1 -17839.109,E2 -17839.109} C_VEL
LIN {X 0,Y 270.276,Z 361.816,A -85,B 0,C 180,E1 -17844.585,E2 -17844.585} C_VEL
LIN {X 0,Y 270.274,Z 361.816,A -85,B 0,C 180,E1 -17847.908,E2 -17847.908} C_VEL
LIN {X 0,Y 270.186,Z 361.829,A -85,B 0,C 180,E1 -17851.348,E2 -17851.348} C_VEL
LIN {X 0,Y 270.217,Z 361.826,A -85,B 0,C 180,E1 -17854.903,E2 -17854.903} C_VEL
LIN {X 0,Y 270.223,Z 361.826,A -85,B 0,C 180,E1 -17858.717,E2 -17858.717} C_VEL
LIN {X 0,Y 270.196,Z 361.827,A -85,B 0,C 180,E1 -17862.553,E2 -17862.553} C_VEL
LIN {X 0,Y 270.172,Z 361.833,A -85,B 0,C 180,E1 -17866.749,E2 -17866.749} C_VEL
LIN {X 0,Y 270.223,Z 361.821,A -85,B 0,C 180,E1 -17871.283,E2 -17871.283} C_VEL
LIN {X 0,Y 270.215,Z 361.824,A -85,B 0,C 180,E1 -17875.096,E2 -17875.096} C_VEL
LIN {X 0,Y 270.201,Z 361.824,A -85,B 0,C 180,E1 -17879.13,E2 -17879.13} C_VEL
LIN {X 0,Y 270.263,Z 361.819,A -85,B 0,C 180,E1 -17882.146,E2 -17882.146} C_VEL
LIN {X 0,Y 270.278,Z 361.815,A -85,B 0,C 180,E1 -17885.519,E2 -17885.519} C_VEL
LIN {X 0,Y 270.304,Z 361.815,A -85,B 0,C 180,E1 -17890.245,E2 -17890.245} C_VEL
LIN {X 0,Y 270.404,Z 361.8,A -85,B 0,C 180,E1 -17894.935,E2 -17894.935} C_VEL
LIN {X 0,Y 270.413,Z 361.799,A -85,B 0,C 180,E1 -17899.518,E2 -17899.518} C_VEL
LIN {X 0,Y 270.599,Z 361.777,A -85,B 0,C 180,E1 -17902.539,E2 -17902.539} C_VEL
LIN {X 0,Y 270.787,Z 361.753,A -85,B 0,C 180,E1 -17908.513,E2 -17908.513} C_VEL
LIN {X 0,Y 270.789,Z 361.753,A -85,B 0,C 180,E1 -17911.487,E2 -17911.487} C_VEL
LIN {X 0,Y 270.599,Z 361.777,A -85,B 0,C 180,E1 -17917.462,E2 -17917.462} C_VEL
LIN {X 0,Y 270.414,Z 361.799,A -85,B 0,C 180,E1 -17920.482,E2 -17920.482} C_VEL
LIN {X 0,Y 270.404,Z 361.8,A -85,B 0,C 180,E1 -17925.065,E2 -17925.065} C_VEL
LIN {X 0,Y 270.303,Z 361.815,A -85,B 0,C 180,E1 -17929.756,E2 -17929.756} C_VEL
LIN {X 0,Y 270.275,Z 361.816,A -85,B 0,C 180,E1 -17934.586,E2 -17934.586} C_VEL
LIN {X 0,Y 270.27,Z 361.818,A -85,B 0,C 180,E1 -17937.909,E2 -17937.909} C_VEL
LIN {X 0,Y 270.185,Z 361.829,A -85,B 0,C 180,E1 -17941.349,E2 -17941.349} C_VEL
LIN {X 0,Y 270.216,Z 361.824,A -85,B 0,C 180,E1 -17944.904,E2 -17944.904} C_VEL
LIN {X 0,Y 270.223,Z 361.821,A -85,B 0,C 180,E1 -17948.717,E2 -17948.717} C_VEL
LIN {X 0,Y 270.249,Z 361.819,A -85,B 0,C 180,E1 -17952.544,E2 -17952.544} C_VEL
LIN {X 0,Y 270.19,Z 361.827,A -85,B 0,C 180,E1 -17956.746,E2 -17956.746} C_VEL
LIN {X 0,Y 270.209,Z 361.827,A -85,B 0,C 180,E1 -17961.375,E2 -17961.375} C_VEL
LIN {X 0,Y 270.204,Z 361.828,A -85,B 0,C 180,E1 -17965.095,E2 -17965.095} C_VEL
LIN {X 0,Y 270.203,Z 361.829,A -85,B 0,C 180,E1 -17969.131,E2 -17969.131} C_VEL
LIN {X 0,Y 270.267,Z 361.817,A -85,B 0,C 180,E1 -17972.146,E2 -17972.146} C_VEL
LIN {X 0,Y 270.28,Z 361.815,A -85,B 0,C 180,E1 -17975.519,E2 -17975.519} C_VEL
LIN {X 0,Y 270.305,Z 361.813,A -85,B 0,C 180,E1 -17980.245,E2 -17980.245} C_VEL
LIN {X 0,Y 270.407,Z 361.803,A -85,B 0,C 180,E1 -17984.936,E2 -17984.936} C_VEL
LIN {X 0,Y 270.446,Z 361.794,A -85,B 0,C 180,E1 -17989.519,E2 -17989.519} C_VEL
LIN {X 0,Y 270.616,Z 361.776,A -85,B 0,C 180,E1 -17992.539,E2 -17992.539} C_VEL
LIN {X 0,Y 270.791,Z 361.755,A -85,B 0,C 180,E1 -17998.513,E2 -17998.513} C_VEL
LIN {X 0,Y 270.792,Z 361.751,A -85,B 0,C 180,E1 -18001.487,E2 -18001.487} C_VEL
LIN {X 0,Y 270.589,Z 361.776,A -85,B 0,C 180,E1 -18007.462,E2 -18007.462} C_VEL
LIN {X 0,Y 270.416,Z 361.802,A -85,B 0,C 180,E1 -18010.482,E2 -18010.482} C_VEL
LIN {X 0,Y 270.407,Z 361.799,A -85,B 0,C 180,E1 -18015.065,E2 -18015.065} C_VEL
LIN {X 0,Y 270.306,Z 361.813,A -85,B 0,C 180,E1 -18019.756,E2 -18019.756} C_VEL
LIN {X 0,Y 270.278,Z 361.815,A -85,B 0,C 180,E1 -18024.585,E2 -18024.585} C_VEL
LIN {X 0,Y 270.274,Z 361.819,A -85,B 0,C 180,E1 -18027.909,E2 -18027.909} C_VEL
LIN {X 0,Y 270.186,Z 361.826,A -85,B 0,C 180,E1 -18030.226,E2 -18030.226} C_VEL
LIN {X 0,Y 269.545,Z 361.91,A -85,B 0,C 180,E1 -18031.47,E2 -18031.47} C_VEL
LIN {X 0,Y 266.764,Z 362.254,A -85,B 0,C 180,E1 -18033.499,E2 -18033.499} C_VEL
LIN {X 0,Y 264.37,Z 362.552,A -85,B 0,C 180,E1 -18035.148,E2 -18035.148} C_VEL
LIN {X 0,Y 263.306,Z 362.686,A -85,B 0,C 180,E1 -18036.424,E2 -18036.424} C_VEL
LIN {X 0,Y 263.199,Z 362.697,A -85,B 0,C 180,E1 -18036.857,E2 -18036.857} C_VEL
LIN {X 0,Y 263.242,Z 362.815,A -85,B 0,C 180,E1 -18041.344,E2 -18041.344} C_VEL
LIN {X 0,Y 264.803,Z 371.09,A -85,B 0,C 180,E1 -18045.774,E2 -18045.774} C_VEL
LIN {X 0,Y 266.464,Z 379.144,A -85,B 0,C 180,E1 -18049.897,E2 -18049.897} C_VEL
LIN {X 0,Y 267.032,Z 382.51,A -85,B 0,C 180,E1 -18051.56,E2 -18051.56} C_VEL
LIN {X 0,Y 266.462,Z 386.777,A -85,B 0,C 180,E1 -18053.598,E2 -18053.598} C_VEL
LIN {X 0,Y 264.793,Z 396.41,A -85,B 0,C 180,E1 -18058.139,E2 -18058.139} C_VEL
LIN {X 0,Y 263.396,Z 406.763,A -85,B 0,C 180,E1 -18063.025,E2 -18063.025} C_VEL
LIN {X 0,Y 262.539,Z 416.412,A -85,B 0,C 180,E1 -18067.575,E2 -18067.575} C_VEL
LIN {X 0,Y 262.511,Z 416.627,A -85,B 0,C 180,E1 -18067.676,E2 -18067.676} C_VEL
LIN {X 0,Y 262.75,Z 429.704,A -85,B 0,C 180,E1 -18068.523,E2 -18068.523} C_VEL
LIN {X 0,Y 263.311,Z 443.172,A -85,B 0,C 180,E1 -18069.697,E2 -18069.697} C_VEL
LIN {X 0,Y 263.979,Z 456.171,A -85,B 0,C 180,E1 -18071.167,E2 -18071.167} C_VEL
LIN {X 0,Y 264.552,Z 467.102,A -85,B 0,C 180,E1 -18072.686,E2 -18072.686} C_VEL
LIN {X 0,Y 264.74,Z 472.869,A -85,B 0,C 180,E1 -18073.617,E2 -18073.617} C_VEL
LIN {X 0,Y 263.719,Z 483.791,A -85,B 0,C 180,E1 -18075.729,E2 -18075.729} C_VEL
LIN {X 0,Y 263.226,Z 491.995,A -85,B 0,C 180,E1 -18077.667,E2 -18077.667} C_VEL
LIN {X 0,Y 262.934,Z 500.001,A -85,B 0,C 180,E1 -18079.994,E2 -18079.994} C_VEL
LIN {X 0,Y 262.983,Z 506.404,A -85,B 0,C 180,E1 -18082.321,E2 -18082.321} C_VEL
LIN {X 0,Y 263.31,Z 511.434,A -85,B 0,C 180,E1 -18084.64,E2 -18084.64} C_VEL
LIN {X 0,Y 263.698,Z 515.184,A -85,B 0,C 180,E1 -18086.944,E2 -18086.944} C_VEL
LIN {X 0,Y 263.856,Z 517.019,A -85,B 0,C 180,E1 -18088.474,E2 -18088.474} C_VEL
LIN {X 0,Y 264.063,Z 518.33,A -85,B 0,C 180,E1 -18090,E2 -18090} C_VEL
LIN {X 0,Y 263.538,Z 519.042,A -85,B 0,C 180,E1 -18091.528,E2 -18091.528} C_VEL
LIN {X 0,Y 263.034,Z 519.337,A -85,B 0,C 180,E1 -18093.063,E2 -18093.063} C_VEL
LIN {X 0,Y 262.608,Z 519.226,A -85,B 0,C 180,E1 -18094.605,E2 -18094.605} C_VEL
LIN {X 0,Y 262.085,Z 518.131,A -85,B 0,C 180,E1 -18097.167,E2 -18097.167} C_VEL
LIN {X 0,Y 261.874,Z 516.434,A -85,B 0,C 180,E1 -18099.266,E2 -18099.266} C_VEL
LIN {X 0,Y 262.263,Z 512.701,A -85,B 0,C 180,E1 -18102.379,E2 -18102.379} C_VEL
LIN {X 0,Y 263.202,Z 508.901,A -85,B 0,C 180,E1 -18104.695,E2 -18104.695} C_VEL
LIN {X 0,Y 265.208,Z 502.66,A -85,B 0,C 180,E1 -18107.663,E2 -18107.663} C_VEL
LIN {X 0,Y 268.047,Z 495.432,A -85,B 0,C 180,E1 -18110.329,E2 -18110.329} C_VEL
LIN {X 0,Y 271.529,Z 486.938,A -85,B 0,C 180,E1 -18112.846,E2 -18112.846} C_VEL
LIN {X 0,Y 274.368,Z 478.471,A -85,B 0,C 180,E1 -18115.002,E2 -18115.002} C_VEL
LIN {X 0,Y 277.581,Z 468.768,A -85,B 0,C 180,E1 -18117.113,E2 -18117.113} C_VEL
LIN {X 0,Y 279.699,Z 459.871,A -85,B 0,C 180,E1 -18118.927,E2 -18118.927} C_VEL
LIN {X 0,Y 281.395,Z 448.38,A -85,B 0,C 180,E1 -18121.255,E2 -18121.255} C_VEL
LIN {X 0,Y 282.22,Z 436.36,A -85,B 0,C 180,E1 -18123.806,E2 -18123.806} C_VEL
LIN {X 0,Y 282.449,Z 424.145,A -85,B 0,C 180,E1 -18126.668,E2 -18126.668} C_VEL
LIN {X 0,Y 282.525,Z 417.35,A -85,B 0,C 180,E1 -18128.455,E2 -18128.455} C_VEL
LIN {X 0,Y 282.647,Z 411.185,A -85,B 0,C 180,E1 -18130.278,E2 -18130.278} C_VEL
LIN {X 0,Y 282.25,Z 408.115,A -85,B 0,C 180,E1 -18131.669,E2 -18131.669} C_VEL
LIN {X 0,Y 281.735,Z 403.984,A -85,B 0,C 180,E1 -18134.305,E2 -18134.305} C_VEL
LIN {X 0,Y 281.726,Z 401.933,A -85,B 0,C 180,E1 -18136.34,E2 -18136.34} C_VEL
LIN {X 0,Y 282.207,Z 400.57,A -85,B 0,C 180,E1 -18138.341,E2 -18138.341} C_VEL
LIN {X 0,Y 283.103,Z 399.886,A -85,B 0,C 180,E1 -18140.316,E2 -18140.316} C_VEL
LIN {X 0,Y 284.271,Z 400.125,A -85,B 0,C 180,E1 -18142.292,E2 -18142.292} C_VEL
LIN {X 0,Y 285.767,Z 401.019,A -85,B 0,C 180,E1 -18144.252,E2 -18144.252} C_VEL
LIN {X 0,Y 287.409,Z 402.895,A -85,B 0,C 180,E1 -18146.243,E2 -18146.243} C_VEL
LIN {X 0,Y 289.229,Z 405.548,A -85,B 0,C 180,E1 -18148.263,E2 -18148.263} C_VEL
LIN {X 0,Y 290.15,Z 407.579,A -85,B 0,C 180,E1 -18149.425,E2 -18149.425} C_VEL
LIN {X 0,Y 290.821,Z 413.037,A -85,B 0,C 180,E1 -18151.611,E2 -18151.611} C_VEL
LIN {X 0,Y 290.908,Z 416.977,A -85,B 0,C 180,E1 -18153.065,E2 -18153.065} C_VEL
LIN {X 0,Y 287.137,Z 425.043,A -85,B 0,C 180,E1 -18154.907,E2 -18154.907} C_VEL
LIN {X 0,Y 283.214,Z 432.456,A -85,B 0,C 180,E1 -18156.993,E2 -18156.993} C_VEL
LIN {X 0,Y 279.244,Z 439.047,A -85,B 0,C 180,E1 -18159.369,E2 -18159.369} C_VEL
LIN {X 0,Y 276.184,Z 443.53,A -85,B 0,C 180,E1 -18161.453,E2 -18161.453} C_VEL
LIN {X 0,Y 273.523,Z 446.994,A -85,B 0,C 180,E1 -18163.582,E2 -18163.582} C_VEL
LIN {X 0,Y 271.88,Z 448.824,A -85,B 0,C 180,E1 -18165.019,E2 -18165.019} C_VEL
LIN {X 0,Y 269.016,Z 451.243,A -85,B 0,C 180,E1 -18167.936,E2 -18167.936} C_VEL
LIN {X 0,Y 266.786,Z 452.163,A -85,B 0,C 180,E1 -18170.905,E2 -18170.905} C_VEL
LIN {X 0,Y 265.15,Z 451.511,A -85,B 0,C 180,E1 -18173.914,E2 -18173.914} C_VEL
LIN {X 0,Y 264.022,Z 449.359,A -85,B 0,C 180,E1 -18176.948,E2 -18176.948} C_VEL
LIN {X 0,Y 263.503,Z 445.559,A -85,B 0,C 180,E1 -18180,E2 -18180} C_VEL
LIN {X 0,Y 263.239,Z 441.634,A -85,B 0,C 180,E1 -18182.295,E2 -18182.295} C_VEL
LIN {X 0,Y 263.094,Z 436.661,A -85,B 0,C 180,E1 -18184.596,E2 -18184.596} C_VEL
LIN {X 0,Y 263.689,Z 429.397,A -85,B 0,C 180,E1 -18187.273,E2 -18187.273} C_VEL
LIN {X 0,Y 264.316,Z 420.774,A -85,B 0,C 180,E1 -18189.794,E2 -18189.794} C_VEL
LIN {X 0,Y 265.041,Z 412.222,A -85,B 0,C 180,E1 -18191.859,E2 -18191.859} C_VEL
LIN {X 0,Y 265.91,Z 401.715,A -85,B 0,C 180,E1 -18193.956,E2 -18193.956} C_VEL
LIN {X 0,Y 266.985,Z 390.127,A -85,B 0,C 180,E1 -18195.849,E2 -18195.849} C_VEL
LIN {X 0,Y 267.593,Z 381.442,A -85,B 0,C 180,E1 -18197.035,E2 -18197.035} C_VEL
LIN {X 0,Y 264.694,Z 368.958,A -85,B 0,C 180,E1 -18198.579,E2 -18198.579} C_VEL
LIN {X 0,Y 263.311,Z 362.708,A -85,B 0,C 180,E1 -18199.236,E2 -18199.236} C_VEL
LIN {X 0,Y 263.228,Z 362.695,A -85,B 0,C 180,E1 -18204.8,E2 -18204.8} C_VEL
LIN {X 0,Y 263.181,Z 362.702,A -85,B 0,C 180,E1 -18208.729,E2 -18208.729} C_VEL
LIN {X 0,Y 263.135,Z 362.705,A -85,B 0,C 180,E1 -18212.288,E2 -18212.288} C_VEL
LIN {X 0,Y 263.19,Z 362.698,A -85,B 0,C 180,E1 -18215.977,E2 -18215.977} C_VEL
LIN {X 0,Y 263.155,Z 362.703,A -85,B 0,C 180,E1 -18219.863,E2 -18219.863} C_VEL
LIN {X 0,Y 263.134,Z 362.704,A -85,B 0,C 180,E1 -18223.981,E2 -18223.981} C_VEL
LIN {X 0,Y 263.126,Z 362.709,A -85,B 0,C 180,E1 -18228.406,E2 -18228.406} C_VEL
LIN {X 0,Y 263.166,Z 362.701,A -85,B 0,C 180,E1 -18232.104,E2 -18232.104} C_VEL
LIN {X 0,Y 263.184,Z 362.7,A -85,B 0,C 180,E1 -18235.89,E2 -18235.89} C_VEL
LIN {X 0,Y 263.148,Z 362.702,A -85,B 0,C 180,E1 -18239.506,E2 -18239.506} C_VEL
LIN {X 0,Y 263.192,Z 362.699,A -85,B 0,C 180,E1 -18243.002,E2 -18243.002} C_VEL
LIN {X 0,Y 263.188,Z 362.702,A -85,B 0,C 180,E1 -18246.387,E2 -18246.387} C_VEL
LIN {X 0,Y 263.27,Z 362.688,A -85,B 0,C 180,E1 -18249.694,E2 -18249.694} C_VEL
LIN {X 0,Y 263.352,Z 362.68,A -85,B 0,C 180,E1 -18254.522,E2 -18254.522} C_VEL
LIN {X 0,Y 263.356,Z 362.677,A -85,B 0,C 180,E1 -18259.234,E2 -18259.234} C_VEL
LIN {X 0,Y 263.559,Z 362.655,A -85,B 0,C 180,E1 -18262.338,E2 -18262.338} C_VEL
LIN {X 0,Y 263.752,Z 362.63,A -85,B 0,C 180,E1 -18268.473,E2 -18268.473} C_VEL
LIN {X 0,Y 263.753,Z 362.63,A -85,B 0,C 180,E1 -18271.527,E2 -18271.527} C_VEL
LIN {X 0,Y 263.559,Z 362.655,A -85,B 0,C 180,E1 -18277.662,E2 -18277.662} C_VEL
LIN {X 0,Y 263.356,Z 362.677,A -85,B 0,C 180,E1 -18280.767,E2 -18280.767} C_VEL
LIN {X 0,Y 263.352,Z 362.68,A -85,B 0,C 180,E1 -18285.478,E2 -18285.478} C_VEL
LIN {X 0,Y 263.265,Z 362.688,A -85,B 0,C 180,E1 -18290.307,E2 -18290.307} C_VEL
LIN {X 0,Y 263.209,Z 362.698,A -85,B 0,C 180,E1 -18295.292,E2 -18295.292} C_VEL
LIN {X 0,Y 263.176,Z 362.699,A -85,B 0,C 180,E1 -18298.73,E2 -18298.73} C_VEL
LIN {X 0,Y 263.134,Z 362.705,A -85,B 0,C 180,E1 -18302.288,E2 -18302.288} C_VEL
LIN {X 0,Y 263.19,Z 362.699,A -85,B 0,C 180,E1 -18305.978,E2 -18305.978} C_VEL
LIN {X 0,Y 263.163,Z 362.702,A -85,B 0,C 180,E1 -18309.863,E2 -18309.863} C_VEL
LIN {X 0,Y 263.207,Z 362.697,A -85,B 0,C 180,E1 -18311.878,E2 -18311.878} C_VEL
LIN {X 0,Y 263.14,Z 362.703,A -85,B 0,C 180,E1 -18316.148,E2 -18316.148} C_VEL
LIN {X 0,Y 263.109,Z 362.708,A -85,B 0,C 180,E1 -18320.128,E2 -18320.128} C_VEL
LIN {X 0,Y 263.164,Z 362.701,A -85,B 0,C 180,E1 -18324.019,E2 -18324.019} C_VEL
LIN {X 0,Y 263.135,Z 362.705,A -85,B 0,C 180,E1 -18327.712,E2 -18327.712} C_VEL
LIN {X 0,Y 263.204,Z 362.696,A -85,B 0,C 180,E1 -18331.783,E2 -18331.783} C_VEL
LIN {X 0,Y 263.229,Z 362.695,A -85,B 0,C 180,E1 -18335.201,E2 -18335.201} C_VEL
LIN {X 0,Y 263.267,Z 362.689,A -85,B 0,C 180,E1 -18339.694,E2 -18339.694} C_VEL
LIN {X 0,Y 263.355,Z 362.679,A -85,B 0,C 180,E1 -18344.522,E2 -18344.522} C_VEL
LIN {X 0,Y 263.378,Z 362.675,A -85,B 0,C 180,E1 -18349.235,E2 -18349.235} C_VEL
LIN {X 0,Y 263.577,Z 362.651,A -85,B 0,C 180,E1 -18352.339,E2 -18352.339} C_VEL
LIN {X 0,Y 263.755,Z 362.632,A -85,B 0,C 180,E1 -18358.473,E2 -18358.473} C_VEL
LIN {X 0,Y 263.756,Z 362.627,A -85,B 0,C 180,E1 -18361.527,E2 -18361.527} C_VEL
LIN {X 0,Y 263.548,Z 362.653,A -85,B 0,C 180,E1 -18367.663,E2 -18367.663} C_VEL
LIN {X 0,Y 263.359,Z 362.679,A -85,B 0,C 180,E1 -18370.766,E2 -18370.766} C_VEL
LIN {X 0,Y 263.355,Z 362.677,A -85,B 0,C 180,E1 -18375.478,E2 -18375.478} C_VEL
LIN {X 0,Y 263.268,Z 362.692,A -85,B 0,C 180,E1 -18380.307,E2 -18380.307} C_VEL
LIN {X 0,Y 263.213,Z 362.694,A -85,B 0,C 180,E1 -18385.291,E2 -18385.291} C_VEL
LIN {X 0,Y 263.17,Z 362.701,A -85,B 0,C 180,E1 -18388.731,E2 -18388.731} C_VEL
LIN {X 0,Y 263.137,Z 362.706,A -85,B 0,C 180,E1 -18392.288,E2 -18392.288} C_VEL
LIN {X 0,Y 263.191,Z 362.702,A -85,B 0,C 180,E1 -18395.978,E2 -18395.978} C_VEL
LIN {X 0,Y 263.199,Z 362.697,A -85,B 0,C 180,E1 -18396.857,E2 -18396.857} C_VEL
LIN {X 0,Y 262.464,Z 362.855,A -85,B 0,C 180,E1 -18397.724,E2 -18397.724} C_VEL
LIN {X 0,Y 259.552,Z 363.152,A -85,B 0,C 180,E1 -18399.086,E2 -18399.086} C_VEL
LIN {X 0,Y 256.787,Z 363.497,A -85,B 0,C 180,E1 -18400.447,E2 -18400.447} C_VEL
LIN {X 0,Y 256.234,Z 363.809,A -85,B 0,C 180,E1 -18401.257,E2 -18401.257} C_VEL
LIN {X 0,Y 256.24,Z 363.864,A -85,B 0,C 180,E1 -18401.29,E2 -18401.29} C_VEL
LIN {X 0,Y 257.895,Z 372.765,A -85,B 0,C 180,E1 -18406.159,E2 -18406.159} C_VEL
LIN {X 0,Y 259.652,Z 381.053,A -85,B 0,C 180,E1 -18410.5,E2 -18410.5} C_VEL
LIN {X 0,Y 259.962,Z 383.284,A -85,B 0,C 180,E1 -18411.629,E2 -18411.629} C_VEL
LIN {X 0,Y 258.992,Z 389.133,A -85,B 0,C 180,E1 -18414.497,E2 -18414.497} C_VEL
LIN {X 0,Y 257.516,Z 397.898,A -85,B 0,C 180,E1 -18418.765,E2 -18418.765} C_VEL
LIN {X 0,Y 256.113,Z 408.55,A -85,B 0,C 180,E1 -18423.956,E2 -18423.956} C_VEL
LIN {X 0,Y 255.481,Z 415.74,A -85,B 0,C 180,E1 -18427.455,E2 -18427.455} C_VEL
LIN {X 0,Y 255.639,Z 428.667,A -85,B 0,C 180,E1 -18428.321,E2 -18428.321} C_VEL
LIN {X 0,Y 256.162,Z 442.059,A -85,B 0,C 180,E1 -18429.524,E2 -18429.524} C_VEL
LIN {X 0,Y 256.81,Z 455.039,A -85,B 0,C 180,E1 -18431.036,E2 -18431.036} C_VEL
LIN {X 0,Y 257.478,Z 467.33,A -85,B 0,C 180,E1 -18432.814,E2 -18432.814} C_VEL
LIN {X 0,Y 257.596,Z 472.99,A -85,B 0,C 180,E1 -18433.782,E2 -18433.782} C_VEL
LIN {X 0,Y 256.703,Z 482.68,A -85,B 0,C 180,E1 -18435.735,E2 -18435.735} C_VEL
LIN {X 0,Y 256.243,Z 490.864,A -85,B 0,C 180,E1 -18437.727,E2 -18437.727} C_VEL
LIN {X 0,Y 255.975,Z 498.851,A -85,B 0,C 180,E1 -18440.119,E2 -18440.119} C_VEL
LIN {X 0,Y 256.018,Z 504.295,A -85,B 0,C 180,E1 -18442.111,E2 -18442.111} C_VEL
LIN {X 0,Y 256.309,Z 509.504,A -85,B 0,C 180,E1 -18444.493,E2 -18444.493} C_VEL
LIN {X 0,Y 256.743,Z 513.438,A -85,B 0,C 180,E1 -18446.862,E2 -18446.862} C_VEL
LIN {X 0,Y 256.914,Z 515.367,A -85,B 0,C 180,E1 -18448.432,E2 -18448.432} C_VEL
LIN {X 0,Y 257.124,Z 516.829,A -85,B 0,C 180,E1 -18450,E2 -18450} C_VEL
LIN {X 0,Y 256.553,Z 517.615,A -85,B 0,C 180,E1 -18451.57,E2 -18451.57} C_VEL
LIN {X 0,Y 256.017,Z 517.979,A -85,B 0,C 180,E1 -18453.147,E2 -18453.147} C_VEL
LIN {X 0,Y 255.232,Z 517.522,A -85,B 0,C 180,E1 -18456.323,E2 -18456.323} C_VEL
LIN {X 0,Y 254.814,Z 515.506,A -85,B 0,C 180,E1 -18459.525,E2 -18459.525} C_VEL
LIN {X 0,Y 255.277,Z 511.99,A -85,B 0,C 180,E1 -18462.724,E2 -18462.724} C_VEL
LIN {X 0,Y 256.757,Z 507.021,A -85,B 0,C 180,E1 -18465.886,E2 -18465.886} C_VEL
LIN {X 0,Y 258.508,Z 502.282,A -85,B 0,C 180,E1 -18468.219,E2 -18468.219} C_VEL
LIN {X 0,Y 261.39,Z 495.594,A -85,B 0,C 180,E1 -18470.87,E2 -18470.87} C_VEL
LIN {X 0,Y 265.017,Z 487.544,A -85,B 0,C 180,E1 -18473.44,E2 -18473.44} C_VEL
LIN {X 0,Y 268.039,Z 479.5,A -85,B 0,C 180,E1 -18475.635,E2 -18475.635} C_VEL
LIN {X 0,Y 271.845,Z 469.022,A -85,B 0,C 180,E1 -18478.059,E2 -18478.059} C_VEL
LIN {X 0,Y 274.158,Z 460.197,A -85,B 0,C 180,E1 -18479.992,E2 -18479.992} C_VEL
LIN {X 0,Y 276.068,Z 449.522,A -85,B 0,C 180,E1 -18482.317,E2 -18482.317} C_VEL
LIN {X 0,Y 277.234,Z 438.583,A -85,B 0,C 180,E1 -18484.824,E2 -18484.824} C_VEL
LIN {X 0,Y 277.942,Z 428.424,A -85,B 0,C 180,E1 -18487.363,E2 -18487.363} C_VEL
LIN {X 0,Y 278.366,Z 422.036,A -85,B 0,C 180,E1 -18489.138,E2 -18489.138} C_VEL
LIN {X 0,Y 278.822,Z 416.22,A -85,B 0,C 180,E1 -18490.947,E2 -18490.947} C_VEL
LIN {X 0,Y 278.455,Z 412.377,A -85,B 0,C 180,E1 -18492.958,E2 -18492.958} C_VEL
LIN {X 0,Y 278.285,Z 409.596,A -85,B 0,C 180,E1 -18495.002,E2 -18495.002} C_VEL
LIN {X 0,Y 278.453,Z 407.713,A -85,B 0,C 180,E1 -18497.05,E2 -18497.05} C_VEL
LIN {X 0,Y 279.054,Z 406.491,A -85,B 0,C 180,E1 -18499.094,E2 -18499.094} C_VEL
LIN {X 0,Y 279.98,Z 406.096,A -85,B 0,C 180,E1 -18501.13,E2 -18501.13} C_VEL
LIN {X 0,Y 281.161,Z 406.54,A -85,B 0,C 180,E1 -18503.136,E2 -18503.136} C_VEL
LIN {X 0,Y 282.589,Z 407.766,A -85,B 0,C 180,E1 -18505.156,E2 -18505.156} C_VEL
LIN {X 0,Y 284.149,Z 409.893,A -85,B 0,C 180,E1 -18507.24,E2 -18507.24} C_VEL
LIN {X 0,Y 285.268,Z 412.185,A -85,B 0,C 180,E1 -18508.844,E2 -18508.844} C_VEL
LIN {X 0,Y 285.68,Z 415.793,A -85,B 0,C 180,E1 -18510.526,E2 -18510.526} C_VEL
LIN {X 0,Y 285.59,Z 420.365,A -85,B 0,C 180,E1 -18512.365,E2 -18512.365} C_VEL
LIN {X 0,Y 281.341,Z 428.497,A -85,B 0,C 180,E1 -18514.353,E2 -18514.353} C_VEL
LIN {X 0,Y 276.606,Z 436.46,A -85,B 0,C 180,E1 -18516.807,E2 -18516.807} C_VEL
LIN {X 0,Y 273.057,Z 441.69,A -85,B 0,C 180,E1 -18518.879,E2 -18518.879} C_VEL
LIN {X 0,Y 268.813,Z 447.054,A -85,B 0,C 180,E1 -18521.715,E2 -18521.715} C_VEL
LIN {X 0,Y 267.02,Z 449.096,A -85,B 0,C 180,E1 -18523.17,E2 -18523.17} C_VEL
LIN {X 0,Y 263.684,Z 451.994,A -85,B 0,C 180,E1 -18526.12,E2 -18526.12} C_VEL
LIN {X 0,Y 261.096,Z 453.37,A -85,B 0,C 180,E1 -18529.139,E2 -18529.139} C_VEL
LIN {X 0,Y 258.967,Z 453.236,A -85,B 0,C 180,E1 -18532.201,E2 -18532.201} C_VEL
LIN {X 0,Y 257.456,Z 451.609,A -85,B 0,C 180,E1 -18535.302,E2 -18535.302} C_VEL
LIN {X 0,Y 256.671,Z 448.357,A -85,B 0,C 180,E1 -18538.431,E2 -18538.431} C_VEL
LIN {X 0,Y 256.279,Z 444.88,A -85,B 0,C 180,E1 -18540.785,E2 -18540.785} C_VEL
LIN {X 0,Y 256.063,Z 440.414,A -85,B 0,C 180,E1 -18543.146,E2 -18543.146} C_VEL
LIN {X 0,Y 256.261,Z 434.852,A -85,B 0,C 180,E1 -18545.508,E2 -18545.508} C_VEL
LIN {X 0,Y 256.711,Z 428.061,A -85,B 0,C 180,E1 -18547.867,E2 -18547.867} C_VEL
LIN {X 0,Y 257.346,Z 419.727,A -85,B 0,C 180,E1 -18550.249,E2 -18550.249} C_VEL
LIN {X 0,Y 258.163,Z 409.773,A -85,B 0,C 180,E1 -18552.579,E2 -18552.579} C_VEL
LIN {X 0,Y 259.093,Z 399.649,A -85,B 0,C 180,E1 -18554.531,E2 -18554.531} C_VEL
LIN {X 0,Y 260.013,Z 388.611,A -85,B 0,C 180,E1 -18556.286,E2 -18556.286} C_VEL
LIN {X 0,Y 260.486,Z 382.97,A -85,B 0,C 180,E1 -18557.062,E2 -18557.062} C_VEL
LIN {X 0,Y 259.25,Z 376.74,A -85,B 0,C 180,E1 -18557.897,E2 -18557.897} C_VEL
LIN {X 0,Y 256.276,Z 363.562,A -85,B 0,C 180,E1 -18559.421,E2 -18559.421} C_VEL
LIN {X 0,Y 256.191,Z 363.572,A -85,B 0,C 180,E1 -18565.138,E2 -18565.138} C_VEL
LIN {X 0,Y 256.116,Z 363.581,A -85,B 0,C 180,E1 -18569.599,E2 -18569.599} C_VEL
LIN {X 0,Y 256.087,Z 363.583,A -85,B 0,C 180,E1 -18573.29,E2 -18573.29} C_VEL
LIN {X 0,Y 256.141,Z 363.578,A -85,B 0,C 180,E1 -18577.278,E2 -18577.278} C_VEL
LIN {X 0,Y 256.085,Z 363.584,A -85,B 0,C 180,E1 -18581.197,E2 -18581.197} C_VEL
LIN {X 0,Y 256.065,Z 363.586,A -85,B 0,C 180,E1 -18585.528,E2 -18585.528} C_VEL
LIN {X 0,Y 256.058,Z 363.59,A -85,B 0,C 180,E1 -18588.797,E2 -18588.797} C_VEL
LIN {X 0,Y 256.146,Z 363.578,A -85,B 0,C 180,E1 -18592.87,E2 -18592.87} C_VEL
LIN {X 0,Y 256.086,Z 363.586,A -85,B 0,C 180,E1 -18596.71,E2 -18596.71} C_VEL
LIN {X 0,Y 256.135,Z 363.576,A -85,B 0,C 180,E1 -18601.406,E2 -18601.406} C_VEL
LIN {X 0,Y 256.169,Z 363.573,A -85,B 0,C 180,E1 -18605.699,E2 -18605.699} C_VEL
LIN {X 0,Y 256.219,Z 363.565,A -85,B 0,C 180,E1 -18609.109,E2 -18609.109} C_VEL
LIN {X 0,Y 256.301,Z 363.56,A -85,B 0,C 180,E1 -18614.085,E2 -18614.085} C_VEL
LIN {X 0,Y 256.298,Z 363.557,A -85,B 0,C 180,E1 -18618.934,E2 -18618.934} C_VEL
LIN {X 0,Y 256.516,Z 363.534,A -85,B 0,C 180,E1 -18622.126,E2 -18622.126} C_VEL
LIN {X 0,Y 256.5,Z 363.531,A -85,B 0,C 180,E1 -18626.859,E2 -18626.859} C_VEL
LIN {X 0,Y 256.766,Z 363.503,A -85,B 0,C 180,E1 -18630,E2 -18630} C_VEL
LIN {X 0,Y 256.501,Z 363.531,A -85,B 0,C 180,E1 -18633.141,E2 -18633.141} C_VEL
LIN {X 0,Y 256.516,Z 363.534,A -85,B 0,C 180,E1 -18637.874,E2 -18637.874} C_VEL
LIN {X 0,Y 256.296,Z 363.555,A -85,B 0,C 180,E1 -18642.672,E2 -18642.672} C_VEL
LIN {X 0,Y 256.284,Z 363.56,A -85,B 0,C 180,E1 -18646.302,E2 -18646.302} C_VEL
LIN {X 0,Y 256.16,Z 363.574,A -85,B 0,C 180,E1 -18651.121,E2 -18651.121} C_VEL
LIN {X 0,Y 256.189,Z 363.572,A -85,B 0,C 180,E1 -18655.139,E2 -18655.139} C_VEL
LIN {X 0,Y 256.112,Z 363.582,A -85,B 0,C 180,E1 -18659.6,E2 -18659.6} C_VEL
LIN {X 0,Y 256.086,Z 363.586,A -85,B 0,C 180,E1 -18663.291,E2 -18663.291} C_VEL
LIN {X 0,Y 256.142,Z 363.58,A -85,B 0,C 180,E1 -18667.279,E2 -18667.279} C_VEL
LIN {X 0,Y 256.132,Z 363.58,A -85,B 0,C 180,E1 -18671.189,E2 -18671.189} C_VEL
LIN {X 0,Y 256.074,Z 363.586,A -85,B 0,C 180,E1 -18675.527,E2 -18675.527} C_VEL
LIN {X 0,Y 256.061,Z 363.587,A -85,B 0,C 180,E1 -18678.798,E2 -18678.798} C_VEL
LIN {X 0,Y 256.132,Z 363.58,A -85,B 0,C 180,E1 -18682.868,E2 -18682.868} C_VEL
LIN {X 0,Y 256.07,Z 363.585,A -85,B 0,C 180,E1 -18686.708,E2 -18686.708} C_VEL
LIN {X 0,Y 256.116,Z 363.581,A -85,B 0,C 180,E1 -18690.401,E2 -18690.401} C_VEL
LIN {X 0,Y 256.191,Z 363.572,A -85,B 0,C 180,E1 -18694.862,E2 -18694.862} C_VEL
LIN {X 0,Y 256.171,Z 363.575,A -85,B 0,C 180,E1 -18699.105,E2 -18699.105} C_VEL
LIN {X 0,Y 256.303,Z 363.555,A -85,B 0,C 180,E1 -18704.086,E2 -18704.086} C_VEL
LIN {X 0,Y 256.314,Z 363.557,A -85,B 0,C 180,E1 -18708.934,E2 -18708.934} C_VEL
LIN {X 0,Y 256.544,Z 363.525,A -85,B 0,C 180,E1 -18712.127,E2 -18712.127} C_VEL
LIN {X 0,Y 256.718,Z 363.508,A -85,B 0,C 180,E1 -18718.432,E2 -18718.432} C_VEL
LIN {X 0,Y 256.719,Z 363.504,A -85,B 0,C 180,E1 -18721.569,E2 -18721.569} C_VEL
LIN {X 0,Y 256.479,Z 363.538,A -85,B 0,C 180,E1 -18726.293,E2 -18726.293} C_VEL
LIN {X 0,Y 256.43,Z 363.539,A -85,B 0,C 180,E1 -18729.465,E2 -18729.465} C_VEL
LIN {X 0,Y 256.26,Z 363.565,A -85,B 0,C 180,E1 -18734.29,E2 -18734.29} C_VEL
LIN {X 0,Y 256.215,Z 363.566,A -85,B 0,C 180,E1 -18737.562,E2 -18737.562} C_VEL
LIN {X 0,Y 256.161,Z 363.574,A -85,B 0,C 180,E1 -18741.12,E2 -18741.12} C_VEL
LIN {X 0,Y 256.192,Z 363.568,A -85,B 0,C 180,E1 -18745.139,E2 -18745.139} C_VEL
LIN {X 0,Y 256.108,Z 363.582,A -85,B 0,C 180,E1 -18749.601,E2 -18749.601} C_VEL
LIN {X 0,Y 256.089,Z 363.583,A -85,B 0,C 180,E1 -18753.29,E2 -18753.29} C_VEL
LIN {X 0,Y 256.132,Z 363.578,A -85,B 0,C 180,E1 -18757.275,E2 -18757.275} C_VEL
LIN {X 0,Y 256.212,Z 363.652,A -85,B 0,C 180,E1 -18761.173,E2 -18761.173} C_VEL
LIN {X 0,Y 256.24,Z 363.864,A -85,B 0,C 180,E1 -18761.29,E2 -18761.29} C_VEL
LIN {X 0,Y 255.914,Z 366.167,A -85,B 0,C 180,E1 -18762.506,E2 -18762.506} C_VEL
LIN {X 0,Y 251.937,Z 373.392,A -85,B 0,C 180,E1 -18766.093,E2 -18766.093} C_VEL
LIN {X 0,Y 251.388,Z 375.771,A -85,B 0,C 180,E1 -18767.33,E2 -18767.33} C_VEL
LIN {X 0,Y 251.468,Z 376.542,A -85,B 0,C 180,E1 -18767.747,E2 -18767.747} C_VEL
LIN {X 0,Y 252.793,Z 382.872,A -85,B 0,C 180,E1 -18771.119,E2 -18771.119} C_VEL
LIN {X 0,Y 252.745,Z 385.133,A -85,B 0,C 180,E1 -18772.284,E2 -18772.284} C_VEL
LIN {X 0,Y 250.928,Z 394.841,A -85,B 0,C 180,E1 -18777.166,E2 -18777.166} C_VEL
LIN {X 0,Y 249.424,Z 405.002,A -85,B 0,C 180,E1 -18782.295,E2 -18782.295} C_VEL
LIN {X 0,Y 248.457,Z 414.746,A -85,B 0,C 180,E1 -18787.221,E2 -18787.221} C_VEL
LIN {X 0,Y 248.572,Z 428.722,A -85,B 0,C 180,E1 -18788.217,E2 -18788.217} C_VEL
LIN {X 0,Y 249.031,Z 441.257,A -85,B 0,C 180,E1 -18789.396,E2 -18789.396} C_VEL
LIN {X 0,Y 249.645,Z 453.738,A -85,B 0,C 180,E1 -18790.897,E2 -18790.897} C_VEL
LIN {X 0,Y 250.332,Z 465.653,A -85,B 0,C 180,E1 -18792.659,E2 -18792.659} C_VEL
LIN {X 0,Y 250.46,Z 472.741,A -85,B 0,C 180,E1 -18793.913,E2 -18793.913} C_VEL
LIN {X 0,Y 249.59,Z 483.266,A -85,B 0,C 180,E1 -18796.152,E2 -18796.152} C_VEL
LIN {X 0,Y 249.116,Z 492.502,A -85,B 0,C 180,E1 -18798.61,E2 -18798.61} C_VEL
LIN {X 0,Y 248.979,Z 500.029,A -85,B 0,C 180,E1 -18801.1,E2 -18801.1} C_VEL
LIN {X 0,Y 249.201,Z 505.843,A -85,B 0,C 180,E1 -18803.523,E2 -18803.523} C_VEL
LIN {X 0,Y 249.667,Z 510.41,A -85,B 0,C 180,E1 -18805.964,E2 -18805.964} C_VEL
LIN {X 0,Y 249.965,Z 513.677,A -85,B 0,C 180,E1 -18808.389,E2 -18808.389} C_VEL
LIN {X 0,Y 250.191,Z 515.224,A -85,B 0,C 180,E1 -18810,E2 -18810} C_VEL
LIN {X 0,Y 249.584,Z 516.126,A -85,B 0,C 180,E1 -18811.614,E2 -18811.614} C_VEL
LIN {X 0,Y 249.025,Z 516.604,A -85,B 0,C 180,E1 -18813.236,E2 -18813.236} C_VEL
LIN {X 0,Y 248.187,Z 516.32,A -85,B 0,C 180,E1 -18816.504,E2 -18816.504} C_VEL
LIN {X 0,Y 247.776,Z 514.502,A -85,B 0,C 180,E1 -18819.799,E2 -18819.799} C_VEL
LIN {X 0,Y 248.31,Z 511.272,A -85,B 0,C 180,E1 -18823.087,E2 -18823.087} C_VEL
LIN {X 0,Y 249.853,Z 506.588,A -85,B 0,C 180,E1 -18826.337,E2 -18826.337} C_VEL
LIN {X 0,Y 252.509,Z 500.403,A -85,B 0,C 180,E1 -18829.511,E2 -18829.511} C_VEL
LIN {X 0,Y 255.808,Z 493.701,A -85,B 0,C 180,E1 -18832.195,E2 -18832.195} C_VEL
LIN {X 0,Y 258.986,Z 486.893,A -85,B 0,C 180,E1 -18834.446,E2 -18834.446} C_VEL
LIN {X 0,Y 262.925,Z 477.712,A -85,B 0,C 180,E1 -18837.027,E2 -18837.027} C_VEL
LIN {X 0,Y 266.371,Z 468.828,A -85,B 0,C 180,E1 -18839.182,E2 -18839.182} C_VEL
LIN {X 0,Y 268.699,Z 460.617,A -85,B 0,C 180,E1 -18841.103,E2 -18841.103} C_VEL
LIN {X 0,Y 270.789,Z 450.897,A -85,B 0,C 180,E1 -18843.382,E2 -18843.382} C_VEL
LIN {X 0,Y 272.348,Z 440.467,A -85,B 0,C 180,E1 -18845.974,E2 -18845.974} C_VEL
LIN {X 0,Y 273.446,Z 431.25,A -85,B 0,C 180,E1 -18848.478,E2 -18848.478} C_VEL
LIN {X 0,Y 274.208,Z 425.065,A -85,B 0,C 180,E1 -18850.365,E2 -18850.365} C_VEL
LIN {X 0,Y 274.848,Z 421.037,A -85,B 0,C 180,E1 -18851.67,E2 -18851.67} C_VEL
LIN {X 0,Y 274.669,Z 416.788,A -85,B 0,C 180,E1 -18854.238,E2 -18854.238} C_VEL
LIN {X 0,Y 274.728,Z 414.502,A -85,B 0,C 180,E1 -18856.314,E2 -18856.314} C_VEL
LIN {X 0,Y 275.097,Z 413.034,A -85,B 0,C 180,E1 -18858.376,E2 -18858.376} C_VEL
LIN {X 0,Y 275.864,Z 412.245,A -85,B 0,C 180,E1 -18860.438,E2 -18860.438} C_VEL
LIN {X 0,Y 276.822,Z 412.321,A -85,B 0,C 180,E1 -18862.46,E2 -18862.46} C_VEL
LIN {X 0,Y 277.986,Z 413.145,A -85,B 0,C 180,E1 -18864.445,E2 -18864.445} C_VEL
LIN {X 0,Y 279.859,Z 415.768,A -85,B 0,C 180,E1 -18867.443,E2 -18867.443} C_VEL
LIN {X 0,Y 280.571,Z 417.848,A -85,B 0,C 180,E1 -18868.91,E2 -18868.91} C_VEL
LIN {X 0,Y 280.474,Z 422.006,A -85,B 0,C 180,E1 -18870.861,E2 -18870.861} C_VEL
LIN {X 0,Y 280.067,Z 424.268,A -85,B 0,C 180,E1 -18871.772,E2 -18871.772} C_VEL
LIN {X 0,Y 275.369,Z 432.303,A -85,B 0,C 180,E1 -18873.879,E2 -18873.879} C_VEL
LIN {X 0,Y 270.594,Z 439.402,A -85,B 0,C 180,E1 -18876.261,E2 -18876.261} C_VEL
LIN {X 0,Y 266.88,Z 444.292,A -85,B 0,C 180,E1 -18878.366,E2 -18878.366} C_VEL
LIN {X 0,Y 263.489,Z 448.196,A -85,B 0,C 180,E1 -18880.524,E2 -18880.524} C_VEL
LIN {X 0,Y 260.529,Z 451.144,A -85,B 0,C 180,E1 -18882.738,E2 -18882.738} C_VEL
LIN {X 0,Y 257.037,Z 453.764,A -85,B 0,C 180,E1 -18885.754,E2 -18885.754} C_VEL
LIN {X 0,Y 254.274,Z 454.813,A -85,B 0,C 180,E1 -18888.844,E2 -18888.844} C_VEL
LIN {X 0,Y 252.047,Z 454.441,A -85,B 0,C 180,E1 -18891.986,E2 -18891.986} C_VEL
LIN {X 0,Y 250.459,Z 452.497,A -85,B 0,C 180,E1 -18895.171,E2 -18895.171} C_VEL
LIN {X 0,Y 249.605,Z 449.029,A -85,B 0,C 180,E1 -18898.386,E2 -18898.386} C_VEL
LIN {X 0,Y 249.191,Z 445.348,A -85,B 0,C 180,E1 -18900.808,E2 -18900.808} C_VEL
LIN {X 0,Y 248.994,Z 440.673,A -85,B 0,C 180,E1 -18903.236,E2 -18903.236} C_VEL
LIN {X 0,Y 249.246,Z 433.784,A -85,B 0,C 180,E1 -18906.069,E2 -18906.069} C_VEL
LIN {X 0,Y 249.886,Z 425.187,A -85,B 0,C 180,E1 -18908.898,E2 -18908.898} C_VEL
LIN {X 0,Y 250.628,Z 416.066,A -85,B 0,C 180,E1 -18911.32,E2 -18911.32} C_VEL
LIN {X 0,Y 251.507,Z 404.956,A -85,B 0,C 180,E1 -18913.74,E2 -18913.74} C_VEL
LIN {X 0,Y 252.6,Z 393.622,A -85,B 0,C 180,E1 -18915.74,E2 -18915.74} C_VEL
LIN {X 0,Y 253.354,Z 382.631,A -85,B 0,C 180,E1 -18917.349,E2 -18917.349} C_VEL
LIN {X 0,Y 250.45,Z 370.287,A -85,B 0,C 180,E1 -18918.937,E2 -18918.937} C_VEL
LIN {X 0,Y 249.225,Z 364.439,A -85,B 0,C 180,E1 -18919.619,E2 -18919.619} C_VEL
LIN {X 0,Y 249.154,Z 364.449,A -85,B 0,C 180,E1 -18925.031,E2 -18925.031} C_VEL
LIN {X 0,Y 249.085,Z 364.459,A -85,B 0,C 180,E1 -18928.993,E2 -18928.993} C_VEL
LIN {X 0,Y 249.038,Z 364.462,A -85,B 0,C 180,E1 -18932.425,E2 -18932.425} C_VEL
LIN {X 0,Y 249.076,Z 364.457,A -85,B 0,C 180,E1 -18936.337,E2 -18936.337} C_VEL
LIN {X 0,Y 249.045,Z 364.462,A -85,B 0,C 180,E1 -18940.47,E2 -18940.47} C_VEL
LIN {X 0,Y 249.012,Z 364.468,A -85,B 0,C 180,E1 -18944.877,E2 -18944.877} C_VEL
LIN {X 0,Y 249.019,Z 364.464,A -85,B 0,C 180,E1 -18947.363,E2 -18947.363} C_VEL
LIN {X 0,Y 249.039,Z 364.459,A -85,B 0,C 180,E1 -18951.622,E2 -18951.622} C_VEL
LIN {X 0,Y 249.062,Z 364.459,A -85,B 0,C 180,E1 -18955.642,E2 -18955.642} C_VEL
LIN {X 0,Y 249.051,Z 364.458,A -85,B 0,C 180,E1 -18959.473,E2 -18959.473} C_VEL
LIN {X 0,Y 249.073,Z 364.457,A -85,B 0,C 180,E1 -18963.162,E2 -18963.162} C_VEL
LIN {X 0,Y 249.086,Z 364.456,A -85,B 0,C 180,E1 -18966.733,E2 -18966.733} C_VEL
LIN {X 0,Y 249.131,Z 364.452,A -85,B 0,C 180,E1 -18970.213,E2 -18970.213} C_VEL
LIN {X 0,Y 249.242,Z 364.437,A -85,B 0,C 180,E1 -18973.622,E2 -18973.622} C_VEL
LIN {X 0,Y 249.245,Z 364.436,A -85,B 0,C 180,E1 -18978.616,E2 -18978.616} C_VEL
LIN {X 0,Y 249.455,Z 364.412,A -85,B 0,C 180,E1 -18981.902,E2 -18981.902} C_VEL
LIN {X 0,Y 249.298,Z 364.427,A -85,B 0,C 180,E1 -18985.149,E2 -18985.149} C_VEL
LIN {X 0,Y 249.677,Z 364.384,A -85,B 0,C 180,E1 -18988.387,E2 -18988.387} C_VEL
LIN {X 0,Y 249.677,Z 364.384,A -85,B 0,C 180,E1 -18991.613,E2 -18991.613} C_VEL
LIN {X 0,Y 249.455,Z 364.41,A -85,B 0,C 180,E1 -18996.471,E2 -18996.471} C_VEL
LIN {X 0,Y 249.344,Z 364.427,A -85,B 0,C 180,E1 -18999.737,E2 -18999.737} C_VEL
LIN {X 0,Y 249.207,Z 364.44,A -85,B 0,C 180,E1 -19004.704,E2 -19004.704} C_VEL
LIN {X 0,Y 249.141,Z 364.45,A -85,B 0,C 180,E1 -19008.077,E2 -19008.077} C_VEL
LIN {X 0,Y 249.089,Z 364.457,A -85,B 0,C 180,E1 -19011.518,E2 -19011.518} C_VEL
LIN {X 0,Y 249.131,Z 364.453,A -85,B 0,C 180,E1 -19015.482,E2 -19015.482} C_VEL
LIN {X 0,Y 249.081,Z 364.456,A -85,B 0,C 180,E1 -19018.992,E2 -19018.992} C_VEL
LIN {X 0,Y 249.037,Z 364.461,A -85,B 0,C 180,E1 -19022.425,E2 -19022.425} C_VEL
LIN {X 0,Y 249.076,Z 364.456,A -85,B 0,C 180,E1 -19026.338,E2 -19026.338} C_VEL
LIN {X 0,Y 249.085,Z 364.455,A -85,B 0,C 180,E1 -19030.463,E2 -19030.463} C_VEL
LIN {X 0,Y 249.075,Z 364.458,A -85,B 0,C 180,E1 -19032.809,E2 -19032.809} C_VEL
LIN {X 0,Y 249.026,Z 364.465,A -85,B 0,C 180,E1 -19037.365,E2 -19037.365} C_VEL
LIN {X 0,Y 249.027,Z 364.464,A -85,B 0,C 180,E1 -19041.62,E2 -19041.62} C_VEL
LIN {X 0,Y 249.045,Z 364.459,A -85,B 0,C 180,E1 -19045.64,E2 -19045.64} C_VEL
LIN {X 0,Y 249.054,Z 364.461,A -85,B 0,C 180,E1 -19049.474,E2 -19049.474} C_VEL
LIN {X 0,Y 249.077,Z 364.457,A -85,B 0,C 180,E1 -19053.163,E2 -19053.163} C_VEL
LIN {X 0,Y 249.083,Z 364.458,A -85,B 0,C 180,E1 -19056.733,E2 -19056.733} C_VEL
LIN {X 0,Y 249.114,Z 364.452,A -85,B 0,C 180,E1 -19060.212,E2 -19060.212} C_VEL
LIN {X 0,Y 249.245,Z 364.434,A -85,B 0,C 180,E1 -19063.622,E2 -19063.622} C_VEL
LIN {X 0,Y 249.257,Z 364.438,A -85,B 0,C 180,E1 -19068.617,E2 -19068.617} C_VEL
LIN {X 0,Y 249.488,Z 364.403,A -85,B 0,C 180,E1 -19071.903,E2 -19071.903} C_VEL
LIN {X 0,Y 249.44,Z 364.414,A -85,B 0,C 180,E1 -19076.77,E2 -19076.77} C_VEL
LIN {X 0,Y 249.732,Z 364.374,A -85,B 0,C 180,E1 -19080,E2 -19080} C_VEL
LIN {X 0,Y 249.44,Z 364.412,A -85,B 0,C 180,E1 -19083.231,E2 -19083.231} C_VEL
LIN {X 0,Y 249.451,Z 364.412,A -85,B 0,C 180,E1 -19086.471,E2 -19086.471} C_VEL
LIN {X 0,Y 249.347,Z 364.422,A -85,B 0,C 180,E1 -19089.737,E2 -19089.737} C_VEL
LIN {X 0,Y 249.21,Z 364.441,A -85,B 0,C 180,E1 -19094.703,E2 -19094.703} C_VEL
LIN {X 0,Y 249.144,Z 364.449,A -85,B 0,C 180,E1 -19098.077,E2 -19098.077} C_VEL
LIN {X 0,Y 249.091,Z 364.456,A -85,B 0,C 180,E1 -19101.518,E2 -19101.518} C_VEL
LIN {X 0,Y 249.135,Z 364.448,A -85,B 0,C 180,E1 -19105.482,E2 -19105.482} C_VEL
LIN {X 0,Y 249.077,Z 364.456,A -85,B 0,C 180,E1 -19108.989,E2 -19108.989} C_VEL
LIN {X 0,Y 249.04,Z 364.461,A -85,B 0,C 180,E1 -19112.425,E2 -19112.425} C_VEL
LIN {X 0,Y 249.073,Z 364.458,A -85,B 0,C 180,E1 -19116.339,E2 -19116.339} C_VEL
LIN {X 0,Y 249.15,Z 364.448,A -85,B 0,C 180,E1 -19120.983,E2 -19120.983} C_VEL
LIN {X 0,Y 250.803,Z 373.382,A -85,B 0,C 180,E1 -19126.018,E2 -19126.018} C_VEL
LIN {X 0,Y 251.468,Z 376.542,A -85,B 0,C 180,E1 -19127.747,E2 -19127.747} C_VEL
LIN {X 0,Y 251.236,Z 378.904,A -85,B 0,C 180,E1 -19128.982,E2 -19128.982} C_VEL
LIN {X 0,Y 249.973,Z 381.333,A -85,B 0,C 180,E1 -19130.193,E2 -19130.193} C_VEL
LIN {X 0,Y 245.415,Z 387.857,A -85,B 0,C 180,E1 -19133.446,E2 -19133.446} C_VEL
LIN {X 0,Y 244.827,Z 389.502,A -85,B 0,C 180,E1 -19134.299,E2 -19134.299} C_VEL
LIN {X 0,Y 243.315,Z 397.895,A -85,B 0,C 180,E1 -19138.673,E2 -19138.673} C_VEL
LIN {X 0,Y 242.083,Z 406.666,A -85,B 0,C 180,E1 -19143.257,E2 -19143.257} C_VEL
LIN {X 0,Y 241.411,Z 413.848,A -85,B 0,C 180,E1 -19147.027,E2 -19147.027} C_VEL
LIN {X 0,Y 241.414,Z 425.982,A -85,B 0,C 180,E1 -19147.892,E2 -19147.892} C_VEL
LIN {X 0,Y 241.81,Z 438.926,A -85,B 0,C 180,E1 -19149.12,E2 -19149.12} C_VEL
LIN {X 0,Y 242.36,Z 450.618,A -85,B 0,C 180,E1 -19150.52,E2 -19150.52} C_VEL
LIN {X 0,Y 243.116,Z 463.168,A -85,B 0,C 180,E1 -19152.389,E2 -19152.389} C_VEL
LIN {X 0,Y 243.482,Z 471.457,A -85,B 0,C 180,E1 -19153.87,E2 -19153.87} C_VEL
LIN {X 0,Y 242.588,Z 481.982,A -85,B 0,C 180,E1 -19156.172,E2 -19156.172} C_VEL
LIN {X 0,Y 242.138,Z 491.231,A -85,B 0,C 180,E1 -19158.701,E2 -19158.701} C_VEL
LIN {X 0,Y 242.048,Z 499.148,A -85,B 0,C 180,E1 -19161.416,E2 -19161.416} C_VEL
LIN {X 0,Y 242.369,Z 505.412,A -85,B 0,C 180,E1 -19164.175,E2 -19164.175} C_VEL
LIN {X 0,Y 242.842,Z 509.761,A -85,B 0,C 180,E1 -19166.682,E2 -19166.682} C_VEL
LIN {X 0,Y 243.039,Z 511.943,A -85,B 0,C 180,E1 -19168.343,E2 -19168.343} C_VEL
LIN {X 0,Y 243.263,Z 513.598,A -85,B 0,C 180,E1 -19170,E2 -19170} C_VEL
LIN {X 0,Y 242.631,Z 514.577,A -85,B 0,C 180,E1 -19171.66,E2 -19171.66} C_VEL
LIN {X 0,Y 242.023,Z 515.132,A -85,B 0,C 180,E1 -19173.329,E2 -19173.329} C_VEL
LIN {X 0,Y 241.132,Z 515.08,A -85,B 0,C 180,E1 -19176.695,E2 -19176.695} C_VEL
LIN {X 0,Y 240.73,Z 513.494,A -85,B 0,C 180,E1 -19180.088,E2 -19180.088} C_VEL
LIN {X 0,Y 241.352,Z 510.496,A -85,B 0,C 180,E1 -19183.471,E2 -19183.471} C_VEL
LIN {X 0,Y 242.989,Z 506.114,A -85,B 0,C 180,E1 -19186.812,E2 -19186.812} C_VEL
LIN {X 0,Y 245.795,Z 500.312,A -85,B 0,C 180,E1 -19190.067,E2 -19190.067} C_VEL
LIN {X 0,Y 249.833,Z 492.927,A -85,B 0,C 180,E1 -19193.193,E2 -19193.193} C_VEL
LIN {X 0,Y 253.088,Z 486.345,A -85,B 0,C 180,E1 -19195.494,E2 -19195.494} C_VEL
LIN {X 0,Y 258.055,Z 476.066,A -85,B 0,C 180,E1 -19198.464,E2 -19198.464} C_VEL
LIN {X 0,Y 261.485,Z 467.321,A -85,B 0,C 180,E1 -19200.708,E2 -19200.708} C_VEL
LIN {X 0,Y 264.685,Z 456.462,A -85,B 0,C 180,E1 -19203.433,E2 -19203.433} C_VEL
LIN {X 0,Y 266.889,Z 446.172,A -85,B 0,C 180,E1 -19206.114,E2 -19206.114} C_VEL
LIN {X 0,Y 268.693,Z 436.4,A -85,B 0,C 180,E1 -19208.885,E2 -19208.885} C_VEL
LIN {X 0,Y 269.862,Z 429.933,A -85,B 0,C 180,E1 -19210.953,E2 -19210.953} C_VEL
LIN {X 0,Y 270.694,Z 425.725,A -85,B 0,C 180,E1 -19212.457,E2 -19212.457} C_VEL
LIN {X 0,Y 270.708,Z 422.547,A -85,B 0,C 180,E1 -19214.504,E2 -19214.504} C_VEL
LIN {X 0,Y 270.86,Z 420.282,A -85,B 0,C 180,E1 -19216.595,E2 -19216.595} C_VEL
LIN {X 0,Y 271.601,Z 418.386,A -85,B 0,C 180,E1 -19219.691,E2 -19219.691} C_VEL
LIN {X 0,Y 272.388,Z 418.073,A -85,B 0,C 180,E1 -19221.739,E2 -19221.739} C_VEL
LIN {X 0,Y 273.343,Z 418.502,A -85,B 0,C 180,E1 -19223.746,E2 -19223.746} C_VEL
LIN {X 0,Y 274.302,Z 419.667,A -85,B 0,C 180,E1 -19225.69,E2 -19225.69} C_VEL
LIN {X 0,Y 275.283,Z 421.369,A -85,B 0,C 180,E1 -19227.579,E2 -19227.579} C_VEL
LIN {X 0,Y 275.61,Z 422.623,A -85,B 0,C 180,E1 -19228.54,E2 -19228.54} C_VEL
LIN {X 0,Y 275.287,Z 425.891,A -85,B 0,C 180,E1 -19230.229,E2 -19230.229} C_VEL
LIN {X 0,Y 275.048,Z 427.411,A -85,B 0,C 180,E1 -19230.955,E2 -19230.955} C_VEL
LIN {X 0,Y 270.373,Z 434.619,A -85,B 0,C 180,E1 -19232.942,E2 -19232.942} C_VEL
LIN {X 0,Y 266.003,Z 440.607,A -85,B 0,C 180,E1 -19234.992,E2 -19234.992} C_VEL
LIN {X 0,Y 261.976,Z 445.51,A -85,B 0,C 180,E1 -19237.108,E2 -19237.108} C_VEL
LIN {X 0,Y 257.166,Z 450.538,A -85,B 0,C 180,E1 -19240.025,E2 -19240.025} C_VEL
LIN {X 0,Y 254.074,Z 453.211,A -85,B 0,C 180,E1 -19242.285,E2 -19242.285} C_VEL
LIN {X 0,Y 250.383,Z 455.466,A -85,B 0,C 180,E1 -19245.367,E2 -19245.367} C_VEL
LIN {X 0,Y 247.476,Z 456.255,A -85,B 0,C 180,E1 -19248.533,E2 -19248.533} C_VEL
LIN {X 0,Y 245.128,Z 455.559,A -85,B 0,C 180,E1 -19251.758,E2 -19251.758} C_VEL
LIN {X 0,Y 243.463,Z 453.366,A -85,B 0,C 180,E1 -19255.032,E2 -19255.032} C_VEL
LIN {X 0,Y 242.693,Z 450.69,A -85,B 0,C 180,E1 -19257.51,E2 -19257.51} C_VEL
LIN {X 0,Y 242.257,Z 447.109,A -85,B 0,C 180,E1 -19260,E2 -19260} C_VEL
LIN {X 0,Y 241.98,Z 442.563,A -85,B 0,C 180,E1 -19262.497,E2 -19262.497} C_VEL
LIN {X 0,Y 241.907,Z 436.931,A -85,B 0,C 180,E1 -19265,E2 -19265} C_VEL
LIN {X 0,Y 242.536,Z 428.809,A -85,B 0,C 180,E1 -19267.911,E2 -19267.911} C_VEL
LIN {X 0,Y 243.15,Z 420.396,A -85,B 0,C 180,E1 -19270.366,E2 -19270.366} C_VEL
LIN {X 0,Y 243.948,Z 411.739,A -85,B 0,C 180,E1 -19272.478,E2 -19272.478} C_VEL
LIN {X 0,Y 244.974,Z 400.511,A -85,B 0,C 180,E1 -19274.75,E2 -19274.75} C_VEL
LIN {X 0,Y 245.997,Z 387.966,A -85,B 0,C 180,E1 -19276.814,E2 -19276.814} C_VEL
LIN {X 0,Y 246.274,Z 383.571,A -85,B 0,C 180,E1 -19277.436,E2 -19277.436} C_VEL
LIN {X 0,Y 243.232,Z 370.385,A -85,B 0,C 180,E1 -19279.165,E2 -19279.165} C_VEL
LIN {X 0,Y 242.173,Z 365.317,A -85,B 0,C 180,E1 -19279.771,E2 -19279.771} C_VEL
LIN {X 0,Y 242.06,Z 365.33,A -85,B 0,C 180,E1 -19283.984,E2 -19283.984} C_VEL
LIN {X 0,Y 242.011,Z 365.337,A -85,B 0,C 180,E1 -19287.687,E2 -19287.687} C_VEL
LIN {X 0,Y 241.978,Z 365.341,A -85,B 0,C 180,E1 -19291.519,E2 -19291.519} C_VEL
LIN {X 0,Y 242.03,Z 365.334,A -85,B 0,C 180,E1 -19295.604,E2 -19295.604} C_VEL
LIN {X 0,Y 241.989,Z 365.339,A -85,B 0,C 180,E1 -19299.712,E2 -19299.712} C_VEL
LIN {X 0,Y 241.94,Z 365.345,A -85,B 0,C 180,E1 -19304.2,E2 -19304.2} C_VEL
LIN {X 0,Y 241.945,Z 365.346,A -85,B 0,C 180,E1 -19308.079,E2 -19308.079} C_VEL
LIN {X 0,Y 242.003,Z 365.338,A -85,B 0,C 180,E1 -19312.42,E2 -19312.42} C_VEL
LIN {X 0,Y 241.992,Z 365.343,A -85,B 0,C 180,E1 -19316.509,E2 -19316.509} C_VEL
LIN {X 0,Y 242.036,Z 365.336,A -85,B 0,C 180,E1 -19320.588,E2 -19320.588} C_VEL
LIN {X 0,Y 242.068,Z 365.332,A -85,B 0,C 180,E1 -19324.183,E2 -19324.183} C_VEL
LIN {X 0,Y 242.065,Z 365.331,A -85,B 0,C 180,E1 -19328.29,E2 -19328.29} C_VEL
LIN {X 0,Y 242.164,Z 365.318,A -85,B 0,C 180,E1 -19333.278,E2 -19333.278} C_VEL
LIN {X 0,Y 242.182,Z 365.318,A -85,B 0,C 180,E1 -19338.28,E2 -19338.28} C_VEL
LIN {X 0,Y 242.401,Z 365.29,A -85,B 0,C 180,E1 -19341.665,E2 -19341.665} C_VEL
LIN {X 0,Y 242.259,Z 365.304,A -85,B 0,C 180,E1 -19345.007,E2 -19345.007} C_VEL
LIN {X 0,Y 242.637,Z 365.261,A -85,B 0,C 180,E1 -19348.34,E2 -19348.34} C_VEL
LIN {X 0,Y 242.638,Z 365.261,A -85,B 0,C 180,E1 -19351.66,E2 -19351.66} C_VEL
LIN {X 0,Y 242.425,Z 365.285,A -85,B 0,C 180,E1 -19356.659,E2 -19356.659} C_VEL
LIN {X 0,Y 242.268,Z 365.307,A -85,B 0,C 180,E1 -19360.024,E2 -19360.024} C_VEL
LIN {X 0,Y 242.168,Z 365.317,A -85,B 0,C 180,E1 -19365.141,E2 -19365.141} C_VEL
LIN {X 0,Y 242.075,Z 365.329,A -85,B 0,C 180,E1 -19368.624,E2 -19368.624} C_VEL
LIN {X 0,Y 242.015,Z 365.336,A -85,B 0,C 180,E1 -19372.18,E2 -19372.18} C_VEL
LIN {X 0,Y 242.067,Z 365.332,A -85,B 0,C 180,E1 -19375.838,E2 -19375.838} C_VEL
LIN {X 0,Y 242.03,Z 365.335,A -85,B 0,C 180,E1 -19379.581,E2 -19379.581} C_VEL
LIN {X 0,Y 241.992,Z 365.343,A -85,B 0,C 180,E1 -19383.491,E2 -19383.491} C_VEL
LIN {X 0,Y 242.014,Z 365.337,A -85,B 0,C 180,E1 -19387.578,E2 -19387.578} C_VEL
LIN {X 0,Y 242,Z 365.339,A -85,B 0,C 180,E1 -19391.91,E2 -19391.91} C_VEL
LIN {X 0,Y 241.945,Z 365.344,A -85,B 0,C 180,E1 -19395.801,E2 -19395.801} C_VEL
LIN {X 0,Y 241.969,Z 365.342,A -85,B 0,C 180,E1 -19400.284,E2 -19400.284} C_VEL
LIN {X 0,Y 241.983,Z 365.34,A -85,B 0,C 180,E1 -19404.489,E2 -19404.489} C_VEL
LIN {X 0,Y 241.977,Z 365.341,A -85,B 0,C 180,E1 -19408.48,E2 -19408.48} C_VEL
LIN {X 0,Y 242.012,Z 365.337,A -85,B 0,C 180,E1 -19412.313,E2 -19412.313} C_VEL
LIN {X 0,Y 242.061,Z 365.33,A -85,B 0,C 180,E1 -19416.017,E2 -19416.017} C_VEL
LIN {X 0,Y 242.041,Z 365.333,A -85,B 0,C 180,E1 -19419.609,E2 -19419.609} C_VEL
LIN {X 0,Y 242.166,Z 365.317,A -85,B 0,C 180,E1 -19423.279,E2 -19423.279} C_VEL
LIN {X 0,Y 242.191,Z 365.316,A -85,B 0,C 180,E1 -19428.28,E2 -19428.28} C_VEL
LIN {X 0,Y 242.439,Z 365.281,A -85,B 0,C 180,E1 -19431.666,E2 -19431.666} C_VEL
LIN {X 0,Y 242.264,Z 365.307,A -85,B 0,C 180,E1 -19435.008,E2 -19435.008} C_VEL
LIN {X 0,Y 242.64,Z 365.261,A -85,B 0,C 180,E1 -19438.34,E2 -19438.34} C_VEL
LIN {X 0,Y 242.641,Z 365.257,A -85,B 0,C 180,E1 -19441.66,E2 -19441.66} C_VEL
LIN {X 0,Y 242.421,Z 365.287,A -85,B 0,C 180,E1 -19446.659,E2 -19446.659} C_VEL
LIN {X 0,Y 242.271,Z 365.305,A -85,B 0,C 180,E1 -19450.024,E2 -19450.024} C_VEL
LIN {X 0,Y 242.171,Z 365.316,A -85,B 0,C 180,E1 -19455.141,E2 -19455.141} C_VEL
LIN {X 0,Y 242.078,Z 365.329,A -85,B 0,C 180,E1 -19458.624,E2 -19458.624} C_VEL
LIN {X 0,Y 242.017,Z 365.34,A -85,B 0,C 180,E1 -19462.18,E2 -19462.18} C_VEL
LIN {X 0,Y 242.07,Z 365.33,A -85,B 0,C 180,E1 -19465.838,E2 -19465.838} C_VEL
LIN {X 0,Y 242.011,Z 365.338,A -85,B 0,C 180,E1 -19469.583,E2 -19469.583} C_VEL
LIN {X 0,Y 241.995,Z 365.339,A -85,B 0,C 180,E1 -19473.491,E2 -19473.491} C_VEL
LIN {X 0,Y 242.009,Z 365.339,A -85,B 0,C 180,E1 -19477.579,E2 -19477.579} C_VEL
LIN {X 0,Y 242.138,Z 365.44,A -85,B 0,C 180,E1 -19480.934,E2 -19480.934} C_VEL
LIN {X 0,Y 243.845,Z 374.586,A -85,B 0,C 180,E1 -19486.233,E2 -19486.233} C_VEL
LIN {X 0,Y 245.525,Z 382.492,A -85,B 0,C 180,E1 -19490.612,E2 -19490.612} C_VEL
LIN {X 0,Y 245.703,Z 385.172,A -85,B 0,C 180,E1 -19492.049,E2 -19492.049} C_VEL
LIN {X 0,Y 244.827,Z 389.502,A -85,B 0,C 180,E1 -19494.299,E2 -19494.299} C_VEL
LIN {X 0,Y 243.687,Z 391.898,A -85,B 0,C 180,E1 -19495.536,E2 -19495.536} C_VEL
LIN {X 0,Y 240.131,Z 395.761,A -85,B 0,C 180,E1 -19497.529,E2 -19497.529} C_VEL
LIN {X 0,Y 237.193,Z 398.822,A -85,B 0,C 180,E1 -19499.156,E2 -19499.156} C_VEL
LIN {X 0,Y 235.775,Z 401.179,A -85,B 0,C 180,E1 -19500.437,E2 -19500.437} C_VEL
LIN {X 0,Y 235.566,Z 401.98,A -85,B 0,C 180,E1 -19500.875,E2 -19500.875} C_VEL
LIN {X 0,Y 234.459,Z 411.62,A -85,B 0,C 180,E1 -19506.129,E2 -19506.129} C_VEL
LIN {X 0,Y 234.359,Z 412.9,A -85,B 0,C 180,E1 -19506.821,E2 -19506.821} C_VEL
LIN {X 0,Y 234.299,Z 425.179,A -85,B 0,C 180,E1 -19507.735,E2 -19507.735} C_VEL
LIN {X 0,Y 234.754,Z 439.591,A -85,B 0,C 180,E1 -19509.175,E2 -19509.175} C_VEL
LIN {X 0,Y 235.371,Z 452.319,A -85,B 0,C 180,E1 -19510.825,E2 -19510.825} C_VEL
LIN {X 0,Y 236.105,Z 463.988,A -85,B 0,C 180,E1 -19512.682,E2 -19512.682} C_VEL
LIN {X 0,Y 236.403,Z 471.135,A -85,B 0,C 180,E1 -19514.038,E2 -19514.038} C_VEL
LIN {X 0,Y 235.62,Z 480.618,A -85,B 0,C 180,E1 -19516.195,E2 -19516.195} C_VEL
LIN {X 0,Y 235.188,Z 489.881,A -85,B 0,C 180,E1 -19518.8,E2 -19518.8} C_VEL
LIN {X 0,Y 235.108,Z 497.341,A -85,B 0,C 180,E1 -19521.404,E2 -19521.404} C_VEL
LIN {X 0,Y 235.402,Z 503.259,A -85,B 0,C 180,E1 -19524.002,E2 -19524.002} C_VEL
LIN {X 0,Y 235.911,Z 507.82,A -85,B 0,C 180,E1 -19526.584,E2 -19526.584} C_VEL
LIN {X 0,Y 236.122,Z 510.109,A -85,B 0,C 180,E1 -19528.294,E2 -19528.294} C_VEL
LIN {X 0,Y 236.346,Z 511.896,A -85,B 0,C 180,E1 -19530,E2 -19530} C_VEL
LIN {X 0,Y 235.671,Z 512.994,A -85,B 0,C 180,E1 -19531.709,E2 -19531.709} C_VEL
LIN {X 0,Y 235.024,Z 513.641,A -85,B 0,C 180,E1 -19533.429,E2 -19533.429} C_VEL
LIN {X 0,Y 234.075,Z 513.761,A -85,B 0,C 180,E1 -19536.898,E2 -19536.898} C_VEL
LIN {X 0,Y 233.707,Z 512.416,A -85,B 0,C 180,E1 -19540.395,E2 -19540.395} C_VEL
LIN {X 0,Y 234.405,Z 509.712,A -85,B 0,C 180,E1 -19543.878,E2 -19543.878} C_VEL
LIN {X 0,Y 236.14,Z 505.627,A -85,B 0,C 180,E1 -19547.315,E2 -19547.315} C_VEL
LIN {X 0,Y 239.13,Z 500.146,A -85,B 0,C 180,E1 -19550.651,E2 -19550.651} C_VEL
LIN {X 0,Y 243.321,Z 493.216,A -85,B 0,C 180,E1 -19553.852,E2 -19553.852} C_VEL
LIN {X 0,Y 247.3,Z 485.892,A -85,B 0,C 180,E1 -19556.59,E2 -19556.59} C_VEL
LIN {X 0,Y 252.587,Z 475.945,A -85,B 0,C 180,E1 -19559.596,E2 -19559.596} C_VEL
LIN {X 0,Y 256.103,Z 467.782,A -85,B 0,C 180,E1 -19561.841,E2 -19561.841} C_VEL
LIN {X 0,Y 259.557,Z 457.397,A -85,B 0,C 180,E1 -19564.654,E2 -19564.654} C_VEL
LIN {X 0,Y 261.908,Z 448.592,A -85,B 0,C 180,E1 -19567.137,E2 -19567.137} C_VEL
LIN {X 0,Y 264.291,Z 438.764,A -85,B 0,C 180,E1 -19570.159,E2 -19570.159} C_VEL
LIN {X 0,Y 265.821,Z 432.78,A -85,B 0,C 180,E1 -19572.244,E2 -19572.244} C_VEL
LIN {X 0,Y 266.276,Z 431.119,A -85,B 0,C 180,E1 -19572.852,E2 -19572.852} C_VEL
LIN {X 0,Y 266.487,Z 428.373,A -85,B 0,C 180,E1 -19574.596,E2 -19574.596} C_VEL
LIN {X 0,Y 266.816,Z 425.44,A -85,B 0,C 180,E1 -19577.522,E2 -19577.522} C_VEL
LIN {X 0,Y 267.395,Z 424.183,A -85,B 0,C 180,E1 -19579.66,E2 -19579.66} C_VEL
LIN {X 0,Y 268.135,Z 423.735,A -85,B 0,C 180,E1 -19581.843,E2 -19581.843} C_VEL
LIN {X 0,Y 269.03,Z 424.194,A -85,B 0,C 180,E1 -19584.08,E2 -19584.08} C_VEL
LIN {X 0,Y 270.168,Z 425.998,A -85,B 0,C 180,E1 -19586.887,E2 -19586.887} C_VEL
LIN {X 0,Y 270.491,Z 426.99,A -85,B 0,C 180,E1 -19587.874,E2 -19587.874} C_VEL
LIN {X 0,Y 270.333,Z 428.841,A -85,B 0,C 180,E1 -19589.085,E2 -19589.085} C_VEL
LIN {X 0,Y 269.54,Z 431.341,A -85,B 0,C 180,E1 -19590.303,E2 -19590.303} C_VEL
LIN {X 0,Y 264.674,Z 438.082,A -85,B 0,C 180,E1 -19592.31,E2 -19592.31} C_VEL
LIN {X 0,Y 260.129,Z 443.673,A -85,B 0,C 180,E1 -19594.388,E2 -19594.388} C_VEL
LIN {X 0,Y 255.905,Z 448.234,A -85,B 0,C 180,E1 -19596.533,E2 -19596.533} C_VEL
LIN {X 0,Y 252.066,Z 451.831,A -85,B 0,C 180,E1 -19598.748,E2 -19598.748} C_VEL
LIN {X 0,Y 249.719,Z 453.729,A -85,B 0,C 180,E1 -19600.261,E2 -19600.261} C_VEL
LIN {X 0,Y 245.568,Z 456.379,A -85,B 0,C 180,E1 -19603.369,E2 -19603.369} C_VEL
LIN {X 0,Y 242.093,Z 457.595,A -85,B 0,C 180,E1 -19606.571,E2 -19606.571} C_VEL
LIN {X 0,Y 239.348,Z 457.318,A -85,B 0,C 180,E1 -19609.852,E2 -19609.852} C_VEL
LIN {X 0,Y 237.236,Z 455.613,A -85,B 0,C 180,E1 -19613.194,E2 -19613.194} C_VEL
LIN {X 0,Y 235.858,Z 452.332,A -85,B 0,C 180,E1 -19616.583,E2 -19616.583} C_VEL
LIN {X 0,Y 235.167,Z 447.503,A -85,B 0,C 180,E1 -19620,E2 -19620} C_VEL
LIN {X 0,Y 234.891,Z 442.734,A -85,B 0,C 180,E1 -19622.572,E2 -19622.572} C_VEL
LIN {X 0,Y 234.996,Z 435.738,A -85,B 0,C 180,E1 -19625.578,E2 -19625.578} C_VEL
LIN {X 0,Y 235.505,Z 428.409,A -85,B 0,C 180,E1 -19628.149,E2 -19628.149} C_VEL
LIN {X 0,Y 236.147,Z 419.756,A -85,B 0,C 180,E1 -19630.664,E2 -19630.664} C_VEL
LIN {X 0,Y 236.958,Z 410.712,A -85,B 0,C 180,E1 -19632.852,E2 -19632.852} C_VEL
LIN {X 0,Y 237.987,Z 399.034,A -85,B 0,C 180,E1 -19635.194,E2 -19635.194} C_VEL
LIN {X 0,Y 238.999,Z 387.319,A -85,B 0,C 180,E1 -19637.101,E2 -19637.101} C_VEL
LIN {X 0,Y 239.228,Z 385.032,A -85,B 0,C 180,E1 -19637.433,E2 -19637.433} C_VEL
LIN {X 0,Y 236.581,Z 373.05,A -85,B 0,C 180,E1 -19639.073,E2 -19639.073} C_VEL
LIN {X 0,Y 235.12,Z 366.195,A -85,B 0,C 180,E1 -19639.877,E2 -19639.877} C_VEL
LIN {X 0,Y 234.99,Z 366.212,A -85,B 0,C 180,E1 -19644.753,E2 -19644.753} C_VEL
LIN {X 0,Y 234.954,Z 366.217,A -85,B 0,C 180,E1 -19648.594,E2 -19648.594} C_VEL
LIN {X 0,Y 234.951,Z 366.217,A -85,B 0,C 180,E1 -19653.117,E2 -19653.117} C_VEL
LIN {X 0,Y 234.947,Z 366.219,A -85,B 0,C 180,E1 -19656.745,E2 -19656.745} C_VEL
LIN {X 0,Y 234.968,Z 366.218,A -85,B 0,C 180,E1 -19658.952,E2 -19658.952} C_VEL
LIN {X 0,Y 234.924,Z 366.218,A -85,B 0,C 180,E1 -19663.477,E2 -19663.477} C_VEL
LIN {X 0,Y 234.891,Z 366.226,A -85,B 0,C 180,E1 -19666.515,E2 -19666.515} C_VEL
LIN {X 0,Y 234.955,Z 366.214,A -85,B 0,C 180,E1 -19671.086,E2 -19671.086} C_VEL
LIN {X 0,Y 234.961,Z 366.215,A -85,B 0,C 180,E1 -19675.367,E2 -19675.367} C_VEL
LIN {X 0,Y 234.969,Z 366.213,A -85,B 0,C 180,E1 -19680.157,E2 -19680.157} C_VEL
LIN {X 0,Y 234.994,Z 366.211,A -85,B 0,C 180,E1 -19683.794,E2 -19683.794} C_VEL
LIN {X 0,Y 235.028,Z 366.205,A -85,B 0,C 180,E1 -19688.971,E2 -19688.971} C_VEL
LIN {X 0,Y 235.097,Z 366.198,A -85,B 0,C 180,E1 -19693.059,E2 -19693.059} C_VEL
LIN {X 0,Y 235.115,Z 366.195,A -85,B 0,C 180,E1 -19697.922,E2 -19697.922} C_VEL
LIN {X 0,Y 235.332,Z 366.169,A -85,B 0,C 180,E1 -19701.412,E2 -19701.412} C_VEL
LIN {X 0,Y 235.375,Z 366.163,A -85,B 0,C 180,E1 -19703.141,E2 -19703.141} C_VEL
LIN {X 0,Y 235.597,Z 366.138,A -85,B 0,C 180,E1 -19708.291,E2 -19708.291} C_VEL
LIN {X 0,Y 235.597,Z 366.138,A -85,B 0,C 180,E1 -19711.71,E2 -19711.71} C_VEL
LIN {X 0,Y 235.375,Z 366.163,A -85,B 0,C 180,E1 -19716.86,E2 -19716.86} C_VEL
LIN {X 0,Y 235.215,Z 366.184,A -85,B 0,C 180,E1 -19720.328,E2 -19720.328} C_VEL
LIN {X 0,Y 235.115,Z 366.198,A -85,B 0,C 180,E1 -19725.607,E2 -19725.607} C_VEL
LIN {X 0,Y 235.01,Z 366.21,A -85,B 0,C 180,E1 -19729.206,E2 -19729.206} C_VEL
LIN {X 0,Y 234.963,Z 366.214,A -85,B 0,C 180,E1 -19732.883,E2 -19732.883} C_VEL
LIN {X 0,Y 234.97,Z 366.214,A -85,B 0,C 180,E1 -19736.658,E2 -19736.658} C_VEL
LIN {X 0,Y 234.933,Z 366.216,A -85,B 0,C 180,E1 -19740.568,E2 -19740.568} C_VEL
LIN {X 0,Y 234.962,Z 366.215,A -85,B 0,C 180,E1 -19744.633,E2 -19744.633} C_VEL
LIN {X 0,Y 234.968,Z 366.213,A -85,B 0,C 180,E1 -19748.952,E2 -19748.952} C_VEL
LIN {X 0,Y 234.976,Z 366.216,A -85,B 0,C 180,E1 -19753.466,E2 -19753.466} C_VEL
LIN {X 0,Y 234.924,Z 366.218,A -85,B 0,C 180,E1 -19756.523,E2 -19756.523} C_VEL
LIN {X 0,Y 234.925,Z 366.223,A -85,B 0,C 180,E1 -19761.08,E2 -19761.08} C_VEL
LIN {X 0,Y 234.929,Z 366.219,A -85,B 0,C 180,E1 -19765.362,E2 -19765.362} C_VEL
LIN {X 0,Y 234.934,Z 366.22,A -85,B 0,C 180,E1 -19769.433,E2 -19769.433} C_VEL
LIN {X 0,Y 234.997,Z 366.208,A -85,B 0,C 180,E1 -19773.794,E2 -19773.794} C_VEL
LIN {X 0,Y 235.015,Z 366.212,A -85,B 0,C 180,E1 -19778.97,E2 -19778.97} C_VEL
LIN {X 0,Y 235.1,Z 366.198,A -85,B 0,C 180,E1 -19783.06,E2 -19783.06} C_VEL
LIN {X 0,Y 235.151,Z 366.192,A -85,B 0,C 180,E1 -19787.924,E2 -19787.924} C_VEL
LIN {X 0,Y 235.394,Z 366.158,A -85,B 0,C 180,E1 -19791.415,E2 -19791.415} C_VEL
LIN {X 0,Y 235.41,Z 366.159,A -85,B 0,C 180,E1 -19793.142,E2 -19793.142} C_VEL
LIN {X 0,Y 235.6,Z 366.138,A -85,B 0,C 180,E1 -19798.291,E2 -19798.291} C_VEL
LIN {X 0,Y 235.6,Z 366.134,A -85,B 0,C 180,E1 -19801.71,E2 -19801.71} C_VEL
LIN {X 0,Y 235.372,Z 366.163,A -85,B 0,C 180,E1 -19806.86,E2 -19806.86} C_VEL
LIN {X 0,Y 235.218,Z 366.185,A -85,B 0,C 180,E1 -19810.328,E2 -19810.328} C_VEL
LIN {X 0,Y 235.118,Z 366.195,A -85,B 0,C 180,E1 -19815.606,E2 -19815.606} C_VEL
LIN {X 0,Y 235.013,Z 366.208,A -85,B 0,C 180,E1 -19819.205,E2 -19819.205} C_VEL
LIN {X 0,Y 234.965,Z 366.214,A -85,B 0,C 180,E1 -19822.883,E2 -19822.883} C_VEL
LIN {X 0,Y 234.972,Z 366.213,A -85,B 0,C 180,E1 -19826.657,E2 -19826.657} C_VEL
LIN {X 0,Y 234.927,Z 366.22,A -85,B 0,C 180,E1 -19830.569,E2 -19830.569} C_VEL
LIN {X 0,Y 234.964,Z 366.213,A -85,B 0,C 180,E1 -19834.633,E2 -19834.633} C_VEL
LIN {X 0,Y 235.044,Z 366.207,A -85,B 0,C 180,E1 -19840.005,E2 -19840.005} C_VEL
LIN {X 0,Y 235.103,Z 366.309,A -85,B 0,C 180,E1 -19840.838,E2 -19840.838} C_VEL
LIN {X 0,Y 236.803,Z 375.368,A -85,B 0,C 180,E1 -19846.245,E2 -19846.245} C_VEL
LIN {X 0,Y 238.259,Z 382.075,A -85,B 0,C 180,E1 -19850.079,E2 -19850.079} C_VEL
LIN {X 0,Y 238.61,Z 385.168,A -85,B 0,C 180,E1 -19851.79,E2 -19851.79} C_VEL
LIN {X 0,Y 237.088,Z 393.153,A -85,B 0,C 180,E1 -19856.1,E2 -19856.1} C_VEL
LIN {X 0,Y 235.566,Z 401.98,A -85,B 0,C 180,E1 -19860.875,E2 -19860.875} C_VEL
LIN {X 0,Y 234.665,Z 403.544,A -85,B 0,C 180,E1 -19861.738,E2 -19861.738} C_VEL
LIN {X 0,Y 231.534,Z 405.892,A -85,B 0,C 180,E1 -19863.083,E2 -19863.083} C_VEL
LIN {X 0,Y 228.407,Z 408.199,A -85,B 0,C 180,E1 -19864.464,E2 -19864.464} C_VEL
LIN {X 0,Y 227.544,Z 409.742,A -85,B 0,C 180,E1 -19865.366,E2 -19865.366} C_VEL
LIN {X 0,Y 227.316,Z 411.911,A -85,B 0,C 180,E1 -19866.601,E2 -19866.601} C_VEL
LIN {X 0,Y 227.257,Z 426.452,A -85,B 0,C 180,E1 -19867.777,E2 -19867.777} C_VEL
LIN {X 0,Y 227.673,Z 439.751,A -85,B 0,C 180,E1 -19869.207,E2 -19869.207} C_VEL
LIN {X 0,Y 228.291,Z 452.224,A -85,B 0,C 180,E1 -19870.907,E2 -19870.907} C_VEL
LIN {X 0,Y 229.047,Z 463.779,A -85,B 0,C 180,E1 -19872.844,E2 -19872.844} C_VEL
LIN {X 0,Y 229.33,Z 470.707,A -85,B 0,C 180,E1 -19874.218,E2 -19874.218} C_VEL
LIN {X 0,Y 228.569,Z 480.848,A -85,B 0,C 180,E1 -19876.667,E2 -19876.667} C_VEL
LIN {X 0,Y 228.198,Z 489.829,A -85,B 0,C 180,E1 -19879.351,E2 -19879.351} C_VEL
LIN {X 0,Y 228.25,Z 497.043,A -85,B 0,C 180,E1 -19882.035,E2 -19882.035} C_VEL
LIN {X 0,Y 228.609,Z 502.722,A -85,B 0,C 180,E1 -19884.708,E2 -19884.708} C_VEL
LIN {X 0,Y 229.116,Z 507.066,A -85,B 0,C 180,E1 -19887.363,E2 -19887.363} C_VEL
LIN {X 0,Y 229.445,Z 510.129,A -85,B 0,C 180,E1 -19890,E2 -19890} C_VEL
LIN {X 0,Y 228.748,Z 511.309,A -85,B 0,C 180,E1 -19891.761,E2 -19891.761} C_VEL
LIN {X 0,Y 228.054,Z 512.066,A -85,B 0,C 180,E1 -19893.534,E2 -19893.534} C_VEL
LIN {X 0,Y 227.017,Z 512.423,A -85,B 0,C 180,E1 -19897.113,E2 -19897.113} C_VEL
LIN {X 0,Y 226.706,Z 511.31,A -85,B 0,C 180,E1 -19900.72,E2 -19900.72} C_VEL
LIN {X 0,Y 227.472,Z 508.851,A -85,B 0,C 180,E1 -19904.31,E2 -19904.31} C_VEL
LIN {X 0,Y 229.314,Z 505.076,A -85,B 0,C 180,E1 -19907.847,E2 -19907.847} C_VEL
LIN {X 0,Y 232.482,Z 499.983,A -85,B 0,C 180,E1 -19911.27,E2 -19911.27} C_VEL
LIN {X 0,Y 236.851,Z 493.449,A -85,B 0,C 180,E1 -19914.546,E2 -19914.546} C_VEL
LIN {X 0,Y 241.649,Z 485.458,A -85,B 0,C 180,E1 -19917.732,E2 -19917.732} C_VEL
LIN {X 0,Y 247.195,Z 475.97,A -85,B 0,C 180,E1 -19920.781,E2 -19920.781} C_VEL
LIN {X 0,Y 250.898,Z 468.069,A -85,B 0,C 180,E1 -19923.107,E2 -19923.107} C_VEL
LIN {X 0,Y 254.473,Z 458.675,A -85,B 0,C 180,E1 -19925.849,E2 -19925.849} C_VEL
LIN {X 0,Y 257.203,Z 450.241,A -85,B 0,C 180,E1 -19928.436,E2 -19928.436} C_VEL
LIN {X 0,Y 259.875,Z 441.67,A -85,B 0,C 180,E1 -19931.268,E2 -19931.268} C_VEL
LIN {X 0,Y 261.817,Z 435.731,A -85,B 0,C 180,E1 -19933.55,E2 -19933.55} C_VEL
LIN {X 0,Y 262.208,Z 432.141,A -85,B 0,C 180,E1 -19936.36,E2 -19936.36} C_VEL
LIN {X 0,Y 262.625,Z 430.422,A -85,B 0,C 180,E1 -19938.53,E2 -19938.53} C_VEL
LIN {X 0,Y 263.274,Z 429.386,A -85,B 0,C 180,E1 -19940.728,E2 -19940.728} C_VEL
LIN {X 0,Y 264.021,Z 429.288,A -85,B 0,C 180,E1 -19942.994,E2 -19942.994} C_VEL
LIN {X 0,Y 264.744,Z 430.172,A -85,B 0,C 180,E1 -19945.381,E2 -19945.381} C_VEL
LIN {X 0,Y 265.334,Z 432.192,A -85,B 0,C 180,E1 -19947.952,E2 -19947.952} C_VEL
LIN {X 0,Y 264.924,Z 433.757,A -85,B 0,C 180,E1 -19948.98,E2 -19948.98} C_VEL
LIN {X 0,Y 264.099,Z 435.233,A -85,B 0,C 180,E1 -19949.628,E2 -19949.628} C_VEL
LIN {X 0,Y 259.043,Z 441.479,A -85,B 0,C 180,E1 -19951.654,E2 -19951.654} C_VEL
LIN {X 0,Y 254.261,Z 446.679,A -85,B 0,C 180,E1 -19953.752,E2 -19953.752} C_VEL
LIN {X 0,Y 249.839,Z 450.893,A -85,B 0,C 180,E1 -19955.928,E2 -19955.928} C_VEL
LIN {X 0,Y 245.842,Z 454.178,A -85,B 0,C 180,E1 -19958.183,E2 -19958.183} C_VEL
LIN {X 0,Y 241.156,Z 457.23,A -85,B 0,C 180,E1 -19961.302,E2 -19961.302} C_VEL
LIN {X 0,Y 237.067,Z 458.823,A -85,B 0,C 180,E1 -19964.525,E2 -19964.525} C_VEL
LIN {X 0,Y 233.834,Z 458.976,A -85,B 0,C 180,E1 -19967.855,E2 -19967.855} C_VEL
LIN {X 0,Y 231.265,Z 457.685,A -85,B 0,C 180,E1 -19971.26,E2 -19971.26} C_VEL
LIN {X 0,Y 229.428,Z 454.892,A -85,B 0,C 180,E1 -19974.727,E2 -19974.727} C_VEL
LIN {X 0,Y 228.582,Z 451.786,A -85,B 0,C 180,E1 -19977.356,E2 -19977.356} C_VEL
LIN {X 0,Y 228.07,Z 447.771,A -85,B 0,C 180,E1 -19980,E2 -19980} C_VEL
LIN {X 0,Y 227.804,Z 442.76,A -85,B 0,C 180,E1 -19982.652,E2 -19982.652} C_VEL
LIN {X 0,Y 227.936,Z 435.527,A -85,B 0,C 180,E1 -19985.751,E2 -19985.751} C_VEL
LIN {X 0,Y 228.482,Z 427.887,A -85,B 0,C 180,E1 -19988.401,E2 -19988.401} C_VEL
LIN {X 0,Y 229.337,Z 417.342,A -85,B 0,C 180,E1 -19991.4,E2 -19991.4} C_VEL
LIN {X 0,Y 230.254,Z 406.417,A -85,B 0,C 180,E1 -19993.908,E2 -19993.908} C_VEL
LIN {X 0,Y 231.401,Z 394.862,A -85,B 0,C 180,E1 -19996.089,E2 -19996.089} C_VEL
LIN {X 0,Y 232.051,Z 385.079,A -85,B 0,C 180,E1 -19997.629,E2 -19997.629} C_VEL
LIN {X 0,Y 229.148,Z 372.378,A -85,B 0,C 180,E1 -19999.38,E2 -19999.38} C_VEL
LIN {X 0,Y 228.042,Z 367.077,A -85,B 0,C 180,E1 -20000.051,E2 -20000.051} C_VEL
LIN {X 0,Y 227.931,Z 367.089,A -85,B 0,C 180,E1 -20005.574,E2 -20005.574} C_VEL
LIN {X 0,Y 227.911,Z 367.094,A -85,B 0,C 180,E1 -20010.296,E2 -20010.296} C_VEL
LIN {X 0,Y 227.891,Z 367.093,A -85,B 0,C 180,E1 -20013.718,E2 -20013.718} C_VEL
LIN {X 0,Y 227.872,Z 367.098,A -85,B 0,C 180,E1 -20018.085,E2 -20018.085} C_VEL
LIN {X 0,Y 227.866,Z 367.099,A -85,B 0,C 180,E1 -20022.729,E2 -20022.729} C_VEL
LIN {X 0,Y 227.817,Z 367.106,A -85,B 0,C 180,E1 -20027.259,E2 -20027.259} C_VEL
LIN {X 0,Y 227.87,Z 367.096,A -85,B 0,C 180,E1 -20031.914,E2 -20031.914} C_VEL
LIN {X 0,Y 227.891,Z 367.099,A -85,B 0,C 180,E1 -20036.373,E2 -20036.373} C_VEL
LIN {X 0,Y 227.919,Z 367.093,A -85,B 0,C 180,E1 -20040.438,E2 -20040.438} C_VEL
LIN {X 0,Y 227.93,Z 367.095,A -85,B 0,C 180,E1 -20044.426,E2 -20044.426} C_VEL
LIN {X 0,Y 227.992,Z 367.084,A -85,B 0,C 180,E1 -20048.29,E2 -20048.29} C_VEL
LIN {X 0,Y 228.036,Z 367.079,A -85,B 0,C 180,E1 -20052.825,E2 -20052.825} C_VEL
LIN {X 0,Y 228.073,Z 367.07,A -85,B 0,C 180,E1 -20057.543,E2 -20057.543} C_VEL
LIN {X 0,Y 228.268,Z 367.049,A -85,B 0,C 180,E1 -20061.145,E2 -20061.145} C_VEL
LIN {X 0,Y 228.325,Z 367.041,A -85,B 0,C 180,E1 -20062.928,E2 -20062.928} C_VEL
LIN {X 0,Y 228.556,Z 367.016,A -85,B 0,C 180,E1 -20068.238,E2 -20068.238} C_VEL
LIN {X 0,Y 228.556,Z 367.016,A -85,B 0,C 180,E1 -20071.762,E2 -20071.762} C_VEL
LIN {X 0,Y 228.325,Z 367.041,A -85,B 0,C 180,E1 -20077.073,E2 -20077.073} C_VEL
LIN {X 0,Y 228.146,Z 367.063,A -85,B 0,C 180,E1 -20080.651,E2 -20080.651} C_VEL
LIN {X 0,Y 228.066,Z 367.074,A -85,B 0,C 180,E1 -20084.272,E2 -20084.272} C_VEL
LIN {X 0,Y 228.004,Z 367.084,A -85,B 0,C 180,E1 -20087.953,E2 -20087.953} C_VEL
LIN {X 0,Y 227.932,Z 367.089,A -85,B 0,C 180,E1 -20092.33,E2 -20092.33} C_VEL
LIN {X 0,Y 227.944,Z 367.089,A -85,B 0,C 180,E1 -20096.603,E2 -20096.603} C_VEL
LIN {X 0,Y 227.909,Z 367.091,A -85,B 0,C 180,E1 -20100.296,E2 -20100.296} C_VEL
LIN {X 0,Y 227.891,Z 367.098,A -85,B 0,C 180,E1 -20103.719,E2 -20103.719} C_VEL
LIN {X 0,Y 227.873,Z 367.095,A -85,B 0,C 180,E1 -20108.086,E2 -20108.086} C_VEL
LIN {X 0,Y 227.918,Z 367.093,A -85,B 0,C 180,E1 -20112.718,E2 -20112.718} C_VEL
LIN {X 0,Y 227.833,Z 367.102,A -85,B 0,C 180,E1 -20117.76,E2 -20117.76} C_VEL
LIN {X 0,Y 227.848,Z 367.101,A -85,B 0,C 180,E1 -20121.91,E2 -20121.91} C_VEL
LIN {X 0,Y 227.881,Z 367.095,A -85,B 0,C 180,E1 -20126.378,E2 -20126.378} C_VEL
LIN {X 0,Y 227.922,Z 367.093,A -85,B 0,C 180,E1 -20130.438,E2 -20130.438} C_VEL
LIN {X 0,Y 227.932,Z 367.089,A -85,B 0,C 180,E1 -20134.426,E2 -20134.426} C_VEL
LIN {X 0,Y 227.965,Z 367.087,A -85,B 0,C 180,E1 -20138.288,E2 -20138.288} C_VEL
LIN {X 0,Y 228.038,Z 367.078,A -85,B 0,C 180,E1 -20142.826,E2 -20142.826} C_VEL
LIN {X 0,Y 228.098,Z 367.07,A -85,B 0,C 180,E1 -20147.545,E2 -20147.545} C_VEL
LIN {X 0,Y 228.329,Z 367.039,A -85,B 0,C 180,E1 -20151.147,E2 -20151.147} C_VEL
LIN {X 0,Y 228.362,Z 367.038,A -85,B 0,C 180,E1 -20152.929,E2 -20152.929} C_VEL
LIN {X 0,Y 228.558,Z 367.014,A -85,B 0,C 180,E1 -20158.238,E2 -20158.238} C_VEL
LIN {X 0,Y 228.559,Z 367.012,A -85,B 0,C 180,E1 -20161.762,E2 -20161.762} C_VEL
LIN {X 0,Y 228.323,Z 367.041,A -85,B 0,C 180,E1 -20167.073,E2 -20167.073} C_VEL
LIN {X 0,Y 228.15,Z 367.065,A -85,B 0,C 180,E1 -20170.651,E2 -20170.651} C_VEL
LIN {X 0,Y 228.069,Z 367.077,A -85,B 0,C 180,E1 -20174.272,E2 -20174.272} C_VEL
LIN {X 0,Y 228.007,Z 367.08,A -85,B 0,C 180,E1 -20177.953,E2 -20177.953} C_VEL
LIN {X 0,Y 227.934,Z 367.093,A -85,B 0,C 180,E1 -20182.33,E2 -20182.33} C_VEL
LIN {X 0,Y 227.946,Z 367.088,A -85,B 0,C 180,E1 -20186.602,E2 -20186.602} C_VEL
LIN {X 0,Y 227.901,Z 367.097,A -85,B 0,C 180,E1 -20190.291,E2 -20190.291} C_VEL
LIN {X 0,Y 227.894,Z 367.096,A -85,B 0,C 180,E1 -20193.718,E2 -20193.718} C_VEL
LIN {X 0,Y 227.892,Z 367.098,A -85,B 0,C 180,E1 -20198.082,E2 -20198.082} C_VEL
LIN {X 0,Y 228.058,Z 367.168,A -85,B 0,C 180,E1 -20200.763,E2 -20200.763} C_VEL
LIN {X 0,Y 229.67,Z 375.818,A -85,B 0,C 180,E1 -20206.085,E2 -20206.085} C_VEL
LIN {X 0,Y 231.268,Z 383.028,A -85,B 0,C 180,E1 -20210.344,E2 -20210.344} C_VEL
LIN {X 0,Y 231.516,Z 384.824,A -85,B 0,C 180,E1 -20211.368,E2 -20211.368} C_VEL
LIN {X 0,Y 230.477,Z 390.581,A -85,B 0,C 180,E1 -20214.593,E2 -20214.593} C_VEL
LIN {X 0,Y 228.867,Z 398.985,A -85,B 0,C 180,E1 -20219.297,E2 -20219.297} C_VEL
LIN {X 0,Y 227.696,Z 408.034,A -85,B 0,C 180,E1 -20224.397,E2 -20224.397} C_VEL
LIN {X 0,Y 227.544,Z 409.742,A -85,B 0,C 180,E1 -20225.366,E2 -20225.366} C_VEL
LIN {X 0,Y 226.945,Z 411.244,A -85,B 0,C 180,E1 -20225.944,E2 -20225.944} C_VEL
LIN {X 0,Y 225.282,Z 413.907,A -85,B 0,C 180,E1 -20226.5,E2 -20226.5} C_VEL
LIN {X 0,Y 221.773,Z 419.62,A -85,B 0,C 180,E1 -20227.114,E2 -20227.114} C_VEL
LIN {X 0,Y 220.461,Z 423.356,A -85,B 0,C 180,E1 -20227.442,E2 -20227.442} C_VEL
LIN {X 0,Y 219.936,Z 429.269,A -85,B 0,C 180,E1 -20228.027,E2 -20228.027} C_VEL
LIN {X 0,Y 220.463,Z 437.057,A -85,B 0,C 180,E1 -20228.911,E2 -20228.911} C_VEL
LIN {X 0,Y 221.103,Z 450.295,A -85,B 0,C 180,E1 -20230.744,E2 -20230.744} C_VEL
LIN {X 0,Y 221.931,Z 462.438,A -85,B 0,C 180,E1 -20232.827,E2 -20232.827} C_VEL
LIN {X 0,Y 222.268,Z 470.148,A -85,B 0,C 180,E1 -20234.409,E2 -20234.409} C_VEL
LIN {X 0,Y 221.608,Z 479.333,A -85,B 0,C 180,E1 -20236.707,E2 -20236.707} C_VEL
LIN {X 0,Y 221.267,Z 488.454,A -85,B 0,C 180,E1 -20239.518,E2 -20239.518} C_VEL
LIN {X 0,Y 221.346,Z 495.589,A -85,B 0,C 180,E1 -20242.244,E2 -20242.244} C_VEL
LIN {X 0,Y 221.658,Z 500.454,A -85,B 0,C 180,E1 -20244.542,E2 -20244.542} C_VEL
LIN {X 0,Y 222.208,Z 505.041,A -85,B 0,C 180,E1 -20247.281,E2 -20247.281} C_VEL
LIN {X 0,Y 222.542,Z 508.298,A -85,B 0,C 180,E1 -20250,E2 -20250} C_VEL
LIN {X 0,Y 221.83,Z 509.6,A -85,B 0,C 180,E1 -20251.815,E2 -20251.815} C_VEL
LIN {X 0,Y 221.101,Z 510.44,A -85,B 0,C 180,E1 -20253.645,E2 -20253.645} C_VEL
LIN {X 0,Y 220.018,Z 510.982,A -85,B 0,C 180,E1 -20257.341,E2 -20257.341} C_VEL
LIN {X 0,Y 219.724,Z 510.128,A -85,B 0,C 180,E1 -20261.064,E2 -20261.064} C_VEL
LIN {X 0,Y 220.558,Z 507.967,A -85,B 0,C 180,E1 -20264.769,E2 -20264.769} C_VEL
LIN {X 0,Y 222.521,Z 504.514,A -85,B 0,C 180,E1 -20268.411,E2 -20268.411} C_VEL
LIN {X 0,Y 225.861,Z 499.754,A -85,B 0,C 180,E1 -20271.925,E2 -20271.925} C_VEL
LIN {X 0,Y 230.425,Z 493.63,A -85,B 0,C 180,E1 -20275.278,E2 -20275.278} C_VEL
LIN {X 0,Y 236.121,Z 485.12,A -85,B 0,C 180,E1 -20278.926,E2 -20278.926} C_VEL
LIN {X 0,Y 241.236,Z 477.22,A -85,B 0,C 180,E1 -20281.628,E2 -20281.628} C_VEL
LIN {X 0,Y 245.724,Z 468.693,A -85,B 0,C 180,E1 -20284.344,E2 -20284.344} C_VEL
LIN {X 0,Y 249.861,Z 459.169,A -85,B 0,C 180,E1 -20287.353,E2 -20287.353} C_VEL
LIN {X 0,Y 253.071,Z 450.644,A -85,B 0,C 180,E1 -20290.217,E2 -20290.217} C_VEL
LIN {X 0,Y 255.863,Z 443.494,A -85,B 0,C 180,E1 -20292.83,E2 -20292.83} C_VEL
LIN {X 0,Y 257.122,Z 440.281,A -85,B 0,C 180,E1 -20294.226,E2 -20294.226} C_VEL
LIN {X 0,Y 257.651,Z 437.056,A -85,B 0,C 180,E1 -20297.005,E2 -20297.005} C_VEL
LIN {X 0,Y 258.236,Z 435.231,A -85,B 0,C 180,E1 -20299.644,E2 -20299.644} C_VEL
